   LIN {X -2.697, Y 24.640, Z 108.800}
   LaserStart_Ext()
   LIN {X 5.542, Y 24.640, Z 108.800}
   LaserEnd_Ext()
   LIN {X 5.139, Y 25.640, Z 108.800}
   LaserStart_Ext()
   LIN {X -2.964, Y 25.640, Z 108.800}
   LaserEnd_Ext()
   LIN {X -3.277, Y 26.640, Z 108.800}
   LaserStart_Ext()
   LIN {X 4.736, Y 26.640, Z 108.800}
   LaserEnd_Ext()
   LIN {X 4.333, Y 27.640, Z 108.800}
   LaserStart_Ext()
   LIN {X -3.590, Y 27.640, Z 108.800}
   LaserEnd_Ext()
   LIN {X -3.904, Y 28.640, Z 108.800}
   LaserStart_Ext()
   LIN {X 3.928, Y 28.640, Z 108.800}
   LaserEnd_Ext()
   LIN {X 3.522, Y 29.640, Z 108.800}
   LaserStart_Ext()
   LIN {X -4.217, Y 29.640, Z 108.800}
   LaserEnd_Ext()
   LIN {X -4.535, Y 30.640, Z 108.800}
   LaserStart_Ext()
   LIN {X 3.115, Y 30.640, Z 108.800}
   LaserEnd_Ext()
   LIN {X 2.665, Y 31.640, Z 108.800}
   LaserStart_Ext()
   LIN {X -4.878, Y 31.640, Z 108.800}
   LaserEnd_Ext()
   LIN {X -5.267, Y 32.640, Z 108.800}
   LaserStart_Ext()
   LIN {X 2.196, Y 32.640, Z 108.800}
   LaserEnd_Ext()
   LIN {X 1.727, Y 33.640, Z 108.800}
   LaserStart_Ext()
   LIN {X -5.672, Y 33.640, Z 108.800}
   LaserEnd_Ext()
   LIN {X -6.078, Y 34.640, Z 108.800}
   LaserStart_Ext()
   LIN {X 1.258, Y 34.640, Z 108.800}
   LaserEnd_Ext()
   LIN {X 0.780, Y 35.640, Z 108.800}
   LaserStart_Ext()
   LIN {X -6.479, Y 35.640, Z 108.800}
   LaserEnd_Ext()
   LIN {X -6.928, Y 36.640, Z 108.800}
   LaserStart_Ext()
   LIN {X 0.261, Y 36.640, Z 108.800}
   LaserEnd_Ext()
   LIN {X -0.257, Y 37.640, Z 108.800}
   LaserStart_Ext()
   LIN {X -7.401, Y 37.640, Z 108.800}
   LaserEnd_Ext()
   LIN {X -7.872, Y 38.640, Z 108.800}
   LaserStart_Ext()
   LIN {X -0.776, Y 38.640, Z 108.800}
   LaserEnd_Ext()
   LIN {X -1.330, Y 39.640, Z 108.800}
   LaserStart_Ext()
   LIN {X -8.360, Y 39.640, Z 108.800}
   LaserEnd_Ext()
   LIN {X -8.875, Y 40.640, Z 108.800}
   LaserStart_Ext()
   LIN {X -1.888, Y 40.640, Z 108.800}
   LaserEnd_Ext()
   LIN {X -2.450, Y 41.640, Z 108.800}
   LaserStart_Ext()
   LIN {X -9.405, Y 41.640, Z 108.800}
   LaserEnd_Ext()
   LIN {X -9.750, Y 42.640, Z 108.800}
   LaserStart_Ext()
   LIN {X -3.040, Y 42.640, Z 108.800}
   LaserEnd_Ext()
   LIN {X -3.637, Y 43.640, Z 108.800}
   LaserStart_Ext()
   LIN {X -9.750, Y 43.640, Z 108.800}
   LaserEnd_Ext()
   LIN {X -9.395, Y 44.640, Z 108.800}
   LaserStart_Ext()
   LIN {X -4.259, Y 44.640, Z 108.800}
   LaserEnd_Ext()
   LIN {X -5.251, Y 45.640, Z 108.800}
   LaserStart_Ext()
   LIN {X -8.233, Y 45.640, Z 108.800}
   LaserEnd_Ext()
   LIN {X 1.489, Y -21.393, Z 109.650}
   LaserStart_Ext()
   LIN {X 0.670, Y -20.523, Z 109.650} C_DIS
   LIN {X 0.063, Y -19.874, Z 109.650} C_DIS
   LIN {X -0.221, Y -19.031, Z 109.650} C_DIS
   LIN {X -0.606, Y -17.898, Z 109.650} C_DIS
   LIN {X -0.326, Y -16.414, Z 109.650} C_DIS
   LIN {X -0.042, Y -14.930, Z 109.650} C_DIS
   LIN {X 0.678, Y -14.083, Z 109.650} C_DIS
   LIN {X 1.314, Y -13.320, Z 109.650} C_DIS
   LIN {X 2.671, Y -12.676, Z 109.650} C_DIS
   LIN {X 3.283, Y -12.391, Z 109.650} C_DIS
   LIN {X 3.733, Y -12.383, Z 109.650} C_DIS
   LIN {X 5.327, Y -12.346, Z 109.650} C_DIS
   LIN {X 7.253, Y -13.170, Z 109.650} C_DIS
   LIN {X 8.910, Y -15.135, Z 109.650} C_DIS
   LIN {X 9.327, Y -17.089, Z 109.650} C_DIS
   LIN {X 9.371, Y -17.296, Z 109.650} C_DIS
   LIN {X 9.327, Y -17.466, Z 109.650} C_DIS
   LIN {X 8.781, Y -19.598, Z 109.650} C_DIS
   LIN {X 7.725, Y -20.854, Z 109.650} C_DIS
   LIN {X 7.412, Y -21.228, Z 109.650} C_DIS
   LIN {X 7.138, Y -21.359, Z 109.650} C_DIS
   LIN {X 5.442, Y -22.155, Z 109.650} C_DIS
   LIN {X 3.827, Y -22.190, Z 109.650} C_DIS
   LIN {X 3.393, Y -22.198, Z 109.650} C_DIS
   LIN {X 2.837, Y -21.962, Z 109.650} C_DIS
   LIN {X 1.489, Y -21.393, Z 109.650}
   LaserEnd_Ext()
   LIN {X -4.282, Y -14.760, Z 109.650}
   LaserStart_Ext()
   LIN {X -3.982, Y -13.681, Z 109.650} C_DIS
   LIN {X -3.420, Y -11.591, Z 109.650} C_DIS
   LIN {X -2.903, Y -9.352, Z 109.650} C_DIS
   LIN {X -2.524, Y -7.491, Z 109.650} C_DIS
   LIN {X -1.956, Y -3.894, Z 109.650} C_DIS
   LIN {X -1.776, Y -2.661, Z 109.650} C_DIS
   LIN {X -1.617, Y 0.191, Z 109.650} C_DIS
   LIN {X -1.266, Y 6.431, Z 109.650} C_DIS
   LIN {X -1.777, Y 13.863, Z 109.650} C_DIS
   LIN {X -1.992, Y 16.194, Z 109.650} C_DIS
   LIN {X -3.301, Y 22.823, Z 109.650} C_DIS
   LIN {X -3.707, Y 24.598, Z 109.650} C_DIS
   LIN {X -5.619, Y 30.703, Z 109.650} C_DIS
   LIN {X -5.779, Y 31.168, Z 109.650} C_DIS
   LIN {X -6.169, Y 32.130, Z 109.650} C_DIS
   LIN {X -7.286, Y 34.920, Z 109.650} C_DIS
   LIN {X -7.746, Y 35.978, Z 109.650} C_DIS
   LIN {X -8.768, Y 38.129, Z 109.650} C_DIS
   LIN {X -9.086, Y 38.790, Z 109.650} C_DIS
   LIN {X -9.358, Y 39.314, Z 109.650} C_DIS
   LIN {X -9.821, Y 40.210, Z 109.650} C_DIS
   LIN {X -10.040, Y 40.622, Z 109.650} C_DIS
   LIN {X -10.410, Y 41.313, Z 109.650} C_DIS
   LIN {X -10.836, Y 42.563, Z 109.650} C_DIS
   LIN {X -10.879, Y 42.690, Z 109.650} C_DIS
   LIN {X -10.870, Y 42.819, Z 109.650} C_DIS
   LIN {X -10.782, Y 44.291, Z 109.650} C_DIS
   LIN {X -10.019, Y 45.769, Z 109.650} C_DIS
   LIN {X -7.883, Y 47.113, Z 109.650} C_DIS
   LIN {X -6.707, Y 47.131, Z 109.650} C_DIS
   LIN {X -6.141, Y 47.141, Z 109.650} C_DIS
   LIN {X -5.839, Y 47.006, Z 109.650} C_DIS
   LIN {X -4.557, Y 46.429, Z 109.650} C_DIS
   LIN {X -3.571, Y 45.353, Z 109.650} C_DIS
   LIN {X -2.779, Y 44.088, Z 109.650} C_DIS
   LIN {X -2.138, Y 43.021, Z 109.650} C_DIS
   LIN {X -1.888, Y 42.601, Z 109.650} C_DIS
   LIN {X -1.451, Y 41.852, Z 109.650} C_DIS
   LIN {X -1.083, Y 41.197, Z 109.650} C_DIS
   LIN {X 0.229, Y 38.835, Z 109.650} C_DIS
   LIN {X 1.364, Y 36.647, Z 109.650} C_DIS
   LIN {X 1.693, Y 36.009, Z 109.650} C_DIS
   LIN {X 2.317, Y 34.705, Z 109.650} C_DIS
   LIN {X 4.029, Y 31.053, Z 109.650} C_DIS
   LIN {X 4.856, Y 29.019, Z 109.650} C_DIS
   LIN {X 6.708, Y 24.426, Z 109.650} C_DIS
   LIN {X 7.270, Y 22.711, Z 109.650} C_DIS
   LIN {X 9.117, Y 17.082, Z 109.650} C_DIS
   LIN {X 10.101, Y 13.078, Z 109.650} C_DIS
   LIN {X 11.511, Y 7.032, Z 109.650} C_DIS
   LIN {X 12.575, Y 0.012, Z 109.650} C_DIS
   LIN {X 12.770, Y -1.347, Z 109.650} C_DIS
   LIN {X 13.254, Y -7.226, Z 109.650} C_DIS
   LIN {X 13.286, Y -7.628, Z 109.650} C_DIS
   LIN {X 13.318, Y -8.447, Z 109.650} C_DIS
   LIN {X 13.422, Y -11.308, Z 109.650} C_DIS
   LIN {X 13.441, Y -14.201, Z 109.650} C_DIS
   LIN {X 13.437, Y -14.410, Z 109.650} C_DIS
   LIN {X 13.375, Y -17.530, Z 109.650} C_DIS
   LIN {X 13.069, Y -19.048, Z 109.650} C_DIS
   LIN {X 12.783, Y -20.433, Z 109.650} C_DIS
   LIN {X 11.737, Y -22.221, Z 109.650} C_DIS
   LIN {X 11.254, Y -23.037, Z 109.650} C_DIS
   LIN {X 10.165, Y -23.855, Z 109.650} C_DIS
   LIN {X 8.463, Y -25.189, Z 109.650} C_DIS
   LIN {X 8.006, Y -25.498, Z 109.650} C_DIS
   LIN {X 6.965, Y -25.798, Z 109.650} C_DIS
   LIN {X 5.376, Y -26.226, Z 109.650} C_DIS
   LIN {X 4.199, Y -26.145, Z 109.650} C_DIS
   LIN {X 2.023, Y -25.999, Z 109.650} C_DIS
   LIN {X -0.563, Y -24.720, Z 109.650} C_DIS
   LIN {X -1.210, Y -24.412, Z 109.650} C_DIS
   LIN {X -1.616, Y -23.929, Z 109.650} C_DIS
   LIN {X -3.645, Y -21.485, Z 109.650} C_DIS
   LIN {X -4.310, Y -19.072, Z 109.650} C_DIS
   LIN {X -4.638, Y -17.911, Z 109.650} C_DIS
   LIN {X -4.449, Y -16.198, Z 109.650} C_DIS
   LIN {X -4.282, Y -14.760, Z 109.650}
   LaserEnd_Ext()
   LIN {X 11.602, Y -20.471, Z 109.650}
   LaserStart_Ext()
   LIN {X 11.602, Y -0.245, Z 109.650}
   LaserEnd_Ext()
   LIN {X 10.602, Y 6.357, Z 109.650}
   LaserStart_Ext()
   LIN {X 10.602, Y -22.175, Z 109.650}
   LaserEnd_Ext()
   LIN {X 9.602, Y -23.027, Z 109.650}
   LaserStart_Ext()
   LIN {X 9.602, Y -20.168, Z 109.650}
   LaserEnd_Ext()
   LIN {X 9.602, Y -14.404, Z 109.650}
   LaserStart_Ext()
   LIN {X 9.602, Y 10.816, Z 109.650}
   LaserEnd_Ext()
   LIN {X 8.602, Y 14.989, Z 109.650}
   LaserStart_Ext()
   LIN {X 8.602, Y -13.204, Z 109.650}
   LaserEnd_Ext()
   LIN {X 8.602, Y -21.365, Z 109.650}
   LaserStart_Ext()
   LIN {X 8.602, Y -23.809, Z 109.650}
   LaserEnd_Ext()
   LIN {X 7.602, Y -24.564, Z 109.650}
   LaserStart_Ext()
   LIN {X 7.602, Y -22.245, Z 109.650}
   LaserEnd_Ext()
   LIN {X 7.602, Y -12.232, Z 109.650}
   LaserStart_Ext()
   LIN {X 7.602, Y 18.492, Z 109.650}
   LaserEnd_Ext()
   LIN {X 6.602, Y 21.540, Z 109.650}
   LaserStart_Ext()
   LIN {X 6.602, Y -11.804, Z 109.650}
   LaserEnd_Ext()
   LIN {X 6.602, Y -22.715, Z 109.650}
   LaserStart_Ext()
   LIN {X 6.602, Y -24.861, Z 109.650}
   LaserEnd_Ext()
   LIN {X 5.602, Y -25.130, Z 109.650}
   LaserStart_Ext()
   LIN {X 5.602, Y -23.141, Z 109.650}
   LaserEnd_Ext()
   LIN {X 5.602, Y -11.386, Z 109.650}
   LaserStart_Ext()
   LIN {X 5.602, Y 24.495, Z 109.650}
   LaserEnd_Ext()
   LIN {X 4.602, Y 26.976, Z 109.650}
   LaserStart_Ext()
   LIN {X 4.602, Y -11.363, Z 109.650}
   LaserEnd_Ext()
   LIN {X 4.602, Y -23.174, Z 109.650}
   LaserStart_Ext()
   LIN {X 4.602, Y -25.171, Z 109.650}
   LaserEnd_Ext()
   LIN {X 3.602, Y -25.103, Z 109.650}
   LaserStart_Ext()
   LIN {X 3.602, Y -23.194, Z 109.650}
   LaserEnd_Ext()
   LIN {X 3.602, Y -11.385, Z 109.650}
   LaserStart_Ext()
   LIN {X 3.602, Y 29.449, Z 109.650}
   LaserEnd_Ext()
   LIN {X 2.602, Y 31.741, Z 109.650}
   LaserStart_Ext()
   LIN {X 2.602, Y -11.605, Z 109.650}
   LaserEnd_Ext()
   LIN {X 2.602, Y -22.948, Z 109.650}
   LaserStart_Ext()
   LIN {X 2.602, Y -25.036, Z 109.650}
   LaserEnd_Ext()
   LIN {X 1.602, Y -24.675, Z 109.650}
   LaserStart_Ext()
   LIN {X 1.602, Y -22.526, Z 109.650}
   LaserEnd_Ext()
   LIN {X 1.602, Y -12.077, Z 109.650}
   LaserStart_Ext()
   LIN {X 1.602, Y 33.874, Z 109.650}
   LaserEnd_Ext()
   LIN {X 0.602, Y 35.943, Z 109.650}
   LaserStart_Ext()
   LIN {X 0.602, Y -12.620, Z 109.650}
   LaserEnd_Ext()
   LIN {X 0.602, Y -21.910, Z 109.650}
   LaserStart_Ext()
   LIN {X 0.602, Y -24.181, Z 109.650}
   LaserEnd_Ext()
   LIN {X -0.398, Y -23.691, Z 109.650}
   LaserStart_Ext()
   LIN {X -0.398, Y -20.845, Z 109.650}
   LaserEnd_Ext()
   LIN {X -0.398, Y -13.805, Z 109.650}
   LaserStart_Ext()
   LIN {X -0.398, Y 4.053, Z 109.650}
   LaserEnd_Ext()
   LIN {X -0.398, Y 8.383, Z 109.650}
   LaserStart_Ext()
   LIN {X -0.398, Y 37.873, Z 109.650}
   LaserEnd_Ext()
   LIN {X -1.398, Y 39.705, Z 109.650}
   LaserStart_Ext()
   LIN {X -1.398, Y 18.348, Z 109.650}
   LaserEnd_Ext()
   LIN {X -1.398, Y -6.770, Z 109.650}
   LaserStart_Ext()
   LIN {X -1.398, Y -16.700, Z 109.650}
   LaserEnd_Ext()
   LIN {X -1.398, Y -18.675, Z 109.650}
   LaserStart_Ext()
   LIN {X -1.398, Y -22.626, Z 109.650}
   LaserEnd_Ext()
   LIN {X -2.398, Y -21.422, Z 109.650}
   LaserStart_Ext()
   LIN {X -2.398, Y -11.608, Z 109.650}
   LaserEnd_Ext()
   LIN {X -2.398, Y 23.362, Z 109.650}
   LaserStart_Ext()
   LIN {X -2.398, Y 41.491, Z 109.650}
   LaserEnd_Ext()
   LIN {X -3.398, Y 43.177, Z 109.650}
   LaserStart_Ext()
   LIN {X -3.398, Y 26.958, Z 109.650}
   LaserEnd_Ext()
   LIN {X -3.398, Y -15.818, Z 109.650}
   LaserStart_Ext()
   LIN {X -3.398, Y -18.623, Z 109.650}
   LaserEnd_Ext()
   LIN {X -4.398, Y 30.150, Z 109.650}
   LaserStart_Ext()
   LIN {X -4.398, Y 44.775, Z 109.650}
   LaserEnd_Ext()
   LIN {X -5.398, Y 45.711, Z 109.650}
   LaserStart_Ext()
   LIN {X -5.398, Y 32.895, Z 109.650}
   LaserEnd_Ext()
   LIN {X -6.398, Y 35.386, Z 109.650}
   LaserStart_Ext()
   LIN {X -6.398, Y 46.137, Z 109.650}
   LaserEnd_Ext()
   LIN {X -7.398, Y 46.120, Z 109.650}
   LaserStart_Ext()
   LIN {X -7.398, Y 37.576, Z 109.650}
   LaserEnd_Ext()
   LIN {X -8.398, Y 39.636, Z 109.650}
   LaserStart_Ext()
   LIN {X -8.398, Y 45.608, Z 109.650}
   LaserEnd_Ext()
   LIN {X -9.398, Y 44.792, Z 109.650}
   LaserStart_Ext()
   LIN {X -9.398, Y 41.541, Z 109.650}
   LaserEnd_Ext()
   LIN {X 9.159, Y -15.876, Z 110.500}
   LaserStart_Ext()
   LIN {X 9.452, Y -17.224, Z 110.500} C_DIS
   LIN {X 8.918, Y -19.313, Z 110.500} C_DIS
   LIN {X 8.863, Y -19.534, Z 110.500} C_DIS
   LIN {X 8.686, Y -19.746, Z 110.500} C_DIS
   LIN {X 7.502, Y -21.161, Z 110.500} C_DIS
   LIN {X 6.049, Y -21.850, Z 110.500} C_DIS
   LIN {X 5.533, Y -22.093, Z 110.500} C_DIS
   LIN {X 4.715, Y -22.110, Z 110.500} C_DIS
   LIN {X 3.485, Y -22.140, Z 110.500} C_DIS
   LIN {X 2.667, Y -21.799, Z 110.500} C_DIS
   LIN {X 1.578, Y -21.339, Z 110.500} C_DIS
   LIN {X 0.585, Y -20.284, Z 110.500} C_DIS
   LIN {X 0.149, Y -19.823, Z 110.500} C_DIS
   LIN {X -0.038, Y -19.279, Z 110.500} C_DIS
   LIN {X -0.524, Y -17.849, Z 110.500} C_DIS
   LIN {X -0.045, Y -15.306, Z 110.500} C_DIS
   LIN {X 0.032, Y -14.881, Z 110.500} C_DIS
   LIN {X 0.198, Y -14.676, Z 110.500} C_DIS
   LIN {X 1.349, Y -13.296, Z 110.500} C_DIS
   LIN {X 2.619, Y -12.693, Z 110.500} C_DIS
   LIN {X 3.324, Y -12.341, Z 110.500} C_DIS
   LIN {X 4.429, Y -12.306, Z 110.500} C_DIS
   LIN {X 5.396, Y -12.284, Z 110.500} C_DIS
   LIN {X 6.103, Y -12.586, Z 110.500} C_DIS
   LIN {X 7.353, Y -13.115, Z 110.500} C_DIS
   LIN {X 8.444, Y -14.415, Z 110.500} C_DIS
   LIN {X 8.985, Y -15.064, Z 110.500} C_DIS
   LIN {X 9.159, Y -15.876, Z 110.500}
   LaserEnd_Ext()
   LIN {X -1.499, Y 1.541, Z 110.500}
   LaserStart_Ext()
   LIN {X -1.737, Y -2.717, Z 110.500} C_DIS
   LIN {X -2.006, Y -4.558, Z 110.500} C_DIS
   LIN {X -2.448, Y -7.354, Z 110.500} C_DIS
   LIN {X -2.950, Y -9.818, Z 110.500} C_DIS
   LIN {X -3.303, Y -11.346, Z 110.500} C_DIS
   LIN {X -4.163, Y -14.551, Z 110.500} C_DIS
   LIN {X -4.207, Y -14.720, Z 110.500} C_DIS
   LIN {X -4.555, Y -17.871, Z 110.500} C_DIS
   LIN {X -3.920, Y -20.117, Z 110.500} C_DIS
   LIN {X -3.554, Y -21.444, Z 110.500} C_DIS
   LIN {X -2.439, Y -22.788, Z 110.500} C_DIS
   LIN {X -1.110, Y -24.364, Z 110.500} C_DIS
   LIN {X 1.005, Y -25.374, Z 110.500} C_DIS
   LIN {X 2.207, Y -25.968, Z 110.500} C_DIS
   LIN {X 3.218, Y -26.036, Z 110.500} C_DIS
   LIN {X 5.323, Y -26.181, Z 110.500} C_DIS
   LIN {X 7.970, Y -25.468, Z 110.500} C_DIS
   LIN {X 8.082, Y -25.440, Z 110.500} C_DIS
   LIN {X 8.193, Y -25.360, Z 110.500} C_DIS
   LIN {X 11.282, Y -23.039, Z 110.500} C_DIS
   LIN {X 12.767, Y -20.530, Z 110.500} C_DIS
   LIN {X 12.871, Y -20.353, Z 110.500} C_DIS
   LIN {X 12.899, Y -20.216, Z 110.500} C_DIS
   LIN {X 13.458, Y -17.448, Z 110.500} C_DIS
   LIN {X 13.500, Y -15.336, Z 110.500} C_DIS
   LIN {X 13.517, Y -14.186, Z 110.500} C_DIS
   LIN {X 13.501, Y -12.892, Z 110.500} C_DIS
   LIN {X 13.490, Y -11.226, Z 110.500} C_DIS
   LIN {X 13.433, Y -9.655, Z 110.500} C_DIS
   LIN {X 13.356, Y -7.714, Z 110.500} C_DIS
   LIN {X 13.282, Y -6.761, Z 110.500} C_DIS
   LIN {X 12.861, Y -1.648, Z 110.500} C_DIS
   LIN {X 12.481, Y 0.998, Z 110.500} C_DIS
   LIN {X 11.630, Y 6.615, Z 110.500} C_DIS
   LIN {X 9.957, Y 13.790, Z 110.500} C_DIS
   LIN {X 9.207, Y 16.842, Z 110.500} C_DIS
   LIN {X 7.168, Y 23.056, Z 110.500} C_DIS
   LIN {X 6.759, Y 24.303, Z 110.500} C_DIS
   LIN {X 4.724, Y 29.352, Z 110.500} C_DIS
   LIN {X 4.151, Y 30.761, Z 110.500} C_DIS
   LIN {X 2.965, Y 33.290, Z 110.500} C_DIS
   LIN {X 1.589, Y 36.165, Z 110.500} C_DIS
   LIN {X 0.864, Y 37.571, Z 110.500} C_DIS
   LIN {X 0.372, Y 38.520, Z 110.500} C_DIS
   LIN {X -0.995, Y 40.981, Z 110.500} C_DIS
   LIN {X -1.347, Y 41.611, Z 110.500} C_DIS
   LIN {X -1.430, Y 41.753, Z 110.500} C_DIS
   LIN {X -2.007, Y 42.738, Z 110.500} C_DIS
   LIN {X -2.678, Y 43.851, Z 110.500} C_DIS
   LIN {X -2.846, Y 44.130, Z 110.500} C_DIS
   LIN {X -2.955, Y 44.305, Z 110.500} C_DIS
   LIN {X -3.637, Y 45.385, Z 110.500} C_DIS
   LIN {X -4.589, Y 46.422, Z 110.500} C_DIS
   LIN {X -4.722, Y 46.507, Z 110.500} C_DIS
   LIN {X -6.216, Y 47.174, Z 110.500} C_DIS
   LIN {X -7.216, Y 47.157, Z 110.500} C_DIS
   LIN {X -7.957, Y 47.142, Z 110.500} C_DIS
   LIN {X -8.723, Y 46.647, Z 110.500} C_DIS
   LIN {X -10.111, Y 45.769, Z 110.500} C_DIS
   LIN {X -10.775, Y 44.442, Z 110.500} C_DIS
   LIN {X -10.858, Y 44.280, Z 110.500} C_DIS
   LIN {X -10.869, Y 44.092, Z 110.500} C_DIS
   LIN {X -10.943, Y 42.710, Z 110.500} C_DIS
   LIN {X -10.569, Y 41.627, Z 110.500} C_DIS
   LIN {X -10.470, Y 41.336, Z 110.500} C_DIS
   LIN {X -10.275, Y 40.974, Z 110.500} C_DIS
   LIN {X -9.878, Y 40.235, Z 110.500} C_DIS
   LIN {X -9.556, Y 39.620, Z 110.500} C_DIS
   LIN {X -9.140, Y 38.817, Z 110.500} C_DIS
   LIN {X -8.066, Y 36.588, Z 110.500} C_DIS
   LIN {X -7.929, Y 36.303, Z 110.500} C_DIS
   LIN {X -7.870, Y 36.182, Z 110.500} C_DIS
   LIN {X -7.812, Y 36.049, Z 110.500} C_DIS
   LIN {X -7.115, Y 34.448, Z 110.500} C_DIS
   LIN {X -5.823, Y 31.221, Z 110.500} C_DIS
   LIN {X -5.719, Y 30.956, Z 110.500} C_DIS
   LIN {X -5.174, Y 29.215, Z 110.500} C_DIS
   LIN {X -3.623, Y 24.264, Z 110.500} C_DIS
   LIN {X -3.378, Y 23.191, Z 110.500} C_DIS
   LIN {X -1.948, Y 15.945, Z 110.500} C_DIS
   LIN {X -1.801, Y 14.356, Z 110.500} C_DIS
   LIN {X -1.239, Y 6.181, Z 110.500} C_DIS
   LIN {X -1.499, Y 1.541, Z 110.500}
   LaserEnd_Ext()
   LIN {X -8.631, Y 45.522, Z 110.500}
   LaserStart_Ext()
   LIN {X -5.120, Y 45.522, Z 110.500}
   LaserEnd_Ext()
   LIN {X -4.275, Y 44.522, Z 110.500}
   LaserStart_Ext()
   LIN {X -9.617, Y 44.522, Z 110.500}
   LaserEnd_Ext()
   LIN {X -9.898, Y 43.522, Z 110.500}
   LaserStart_Ext()
   LIN {X -3.647, Y 43.522, Z 110.500}
   LaserEnd_Ext()
   LIN {X -3.044, Y 42.522, Z 110.500}
   LaserStart_Ext()
   LIN {X -9.820, Y 42.522, Z 110.500}
   LaserEnd_Ext()
   LIN {X -9.434, Y 41.522, Z 110.500}
   LaserStart_Ext()
   LIN {X -2.454, Y 41.522, Z 110.500}
   LaserEnd_Ext()
   LIN {X -1.884, Y 40.522, Z 110.500}
   LaserStart_Ext()
   LIN {X -8.899, Y 40.522, Z 110.500}
   LaserEnd_Ext()
   LIN {X -8.379, Y 39.522, Z 110.500}
   LaserStart_Ext()
   LIN {X -1.328, Y 39.522, Z 110.500}
   LaserEnd_Ext()
   LIN {X -0.773, Y 38.522, Z 110.500}
   LaserStart_Ext()
   LIN {X -7.888, Y 38.522, Z 110.500}
   LaserEnd_Ext()
   LIN {X -7.406, Y 37.522, Z 110.500}
   LaserStart_Ext()
   LIN {X -0.236, Y 37.522, Z 110.500}
   LaserEnd_Ext()
   LIN {X 0.280, Y 36.522, Z 110.500}
   LaserStart_Ext()
   LIN {X -6.927, Y 36.522, Z 110.500}
   LaserEnd_Ext()
   LIN {X -6.492, Y 35.522, Z 110.500}
   LaserStart_Ext()
   LIN {X 0.788, Y 35.522, Z 110.500}
   LaserEnd_Ext()
   LIN {X 1.267, Y 34.522, Z 110.500}
   LaserStart_Ext()
   LIN {X -6.067, Y 34.522, Z 110.500}
   LaserEnd_Ext()
   LIN {X -5.667, Y 33.522, Z 110.500}
   LaserStart_Ext()
   LIN {X 1.745, Y 33.522, Z 110.500}
   LaserEnd_Ext()
   LIN {X 2.220, Y 32.522, Z 110.500}
   LaserStart_Ext()
   LIN {X -5.267, Y 32.522, Z 110.500}
   LaserEnd_Ext()
   LIN {X -4.867, Y 31.522, Z 110.500}
   LaserStart_Ext()
   LIN {X 2.689, Y 31.522, Z 110.500}
   LaserEnd_Ext()
   LIN {X 3.158, Y 30.522, Z 110.500}
   LaserStart_Ext()
   LIN {X -4.533, Y 30.522, Z 110.500}
   LaserEnd_Ext()
   LIN {X -4.223, Y 29.522, Z 110.500}
   LaserStart_Ext()
   LIN {X 3.575, Y 29.522, Z 110.500}
   LaserEnd_Ext()
   LIN {X 3.980, Y 28.522, Z 110.500}
   LaserStart_Ext()
   LIN {X -3.909, Y 28.522, Z 110.500}
   LaserEnd_Ext()
   LIN {X -3.596, Y 27.522, Z 110.500}
   LaserStart_Ext()
   LIN {X 4.383, Y 27.522, Z 110.500}
   LaserEnd_Ext()
   LIN {X 4.787, Y 26.522, Z 110.500}
   LaserStart_Ext()
   LIN {X -3.283, Y 26.522, Z 110.500}
   LaserEnd_Ext()
   LIN {X -2.969, Y 25.522, Z 110.500}
   LaserStart_Ext()
   LIN {X 5.190, Y 25.522, Z 110.500}
   LaserEnd_Ext()
   LIN {X 5.593, Y 24.522, Z 110.500}
   LaserStart_Ext()
   LIN {X -2.658, Y 24.522, Z 110.500}
   LaserEnd_Ext()
   LIN {X -2.428, Y 23.522, Z 110.500}
   LaserStart_Ext()
   LIN {X 5.963, Y 23.522, Z 110.500}
   LaserEnd_Ext()
   LIN {X 6.291, Y 22.522, Z 110.500}
   LaserStart_Ext()
   LIN {X -2.226, Y 22.522, Z 110.500}
   LaserEnd_Ext()
   LIN {X -2.029, Y 21.522, Z 110.500}
   LaserStart_Ext()
   LIN {X 6.619, Y 21.522, Z 110.500}
   LaserEnd_Ext()
   LIN {X 6.947, Y 20.522, Z 110.500}
   LaserStart_Ext()
   LIN {X -1.832, Y 20.522, Z 110.500}
   LaserEnd_Ext()
   LIN {X -1.634, Y 19.522, Z 110.500}
   LaserStart_Ext()
   LIN {X 7.275, Y 19.522, Z 110.500}
   LaserEnd_Ext()
   LIN {X 7.603, Y 18.522, Z 110.500}
   LaserStart_Ext()
   LIN {X -1.437, Y 18.522, Z 110.500}
   LaserEnd_Ext()
   LIN {X -1.240, Y 17.522, Z 110.500}
   LaserStart_Ext()
   LIN {X 7.931, Y 17.522, Z 110.500}
   LaserEnd_Ext()
   LIN {X 8.256, Y 16.522, Z 110.500}
   LaserStart_Ext()
   LIN {X -1.042, Y 16.522, Z 110.500}
   LaserEnd_Ext()
   LIN {X -0.904, Y 15.522, Z 110.500}
   LaserStart_Ext()
   LIN {X 8.502, Y 15.522, Z 110.500}
   LaserEnd_Ext()
   LIN {X 8.747, Y 14.522, Z 110.500}
   LaserStart_Ext()
   LIN {X -0.812, Y 14.522, Z 110.500}
   LaserEnd_Ext()
   LIN {X -0.741, Y 13.522, Z 110.500}
   LaserStart_Ext()
   LIN {X 8.993, Y 13.522, Z 110.500}
   LaserEnd_Ext()
   LIN {X 9.226, Y 12.522, Z 110.500}
   LaserStart_Ext()
   LIN {X -0.673, Y 12.522, Z 110.500}
   LaserEnd_Ext()
   LIN {X -0.604, Y 11.522, Z 110.500}
   LaserStart_Ext()
   LIN {X 9.459, Y 11.522, Z 110.500}
   LaserEnd_Ext()
   LIN {X 9.692, Y 10.522, Z 110.500}
   LaserStart_Ext()
   LIN {X -0.535, Y 10.522, Z 110.500}
   LaserEnd_Ext()
   LIN {X -0.466, Y 9.522, Z 110.500}
   LaserStart_Ext()
   LIN {X 9.925, Y 9.522, Z 110.500}
   LaserEnd_Ext()
   LIN {X 10.159, Y 8.522, Z 110.500}
   LaserStart_Ext()
   LIN {X -0.397, Y 8.522, Z 110.500}
   LaserEnd_Ext()
   LIN {X -0.329, Y 7.522, Z 110.500}
   LaserStart_Ext()
   LIN {X 10.392, Y 7.522, Z 110.500}
   LaserEnd_Ext()
   LIN {X 10.625, Y 6.522, Z 110.500}
   LaserStart_Ext()
   LIN {X -0.260, Y 6.522, Z 110.500}
   LaserEnd_Ext()
   LIN {X -0.274, Y 5.522, Z 110.500}
   LaserStart_Ext()
   LIN {X 10.784, Y 5.522, Z 110.500}
   LaserEnd_Ext()
   LIN {X 10.936, Y 4.522, Z 110.500}
   LaserStart_Ext()
   LIN {X -0.330, Y 4.522, Z 110.500}
   LaserEnd_Ext()
   LIN {X -0.386, Y 3.522, Z 110.500}
   LaserStart_Ext()
   LIN {X 11.087, Y 3.522, Z 110.500}
   LaserEnd_Ext()
   LIN {X 11.239, Y 2.522, Z 110.500}
   LaserStart_Ext()
   LIN {X -0.443, Y 2.522, Z 110.500}
   LaserEnd_Ext()
   LIN {X -0.499, Y 1.522, Z 110.500}
   LaserStart_Ext()
   LIN {X 11.391, Y 1.522, Z 110.500}
   LaserEnd_Ext()
   LIN {X 11.540, Y 0.522, Z 110.500}
   LaserStart_Ext()
   LIN {X -0.555, Y 0.522, Z 110.500}
   LaserEnd_Ext()
   LIN {X -0.610, Y -0.478, Z 110.500}
   LaserStart_Ext()
   LIN {X 11.683, Y -0.478, Z 110.500}
   LaserEnd_Ext()
   LIN {X 11.826, Y -1.478, Z 110.500}
   LaserStart_Ext()
   LIN {X -0.666, Y -1.478, Z 110.500}
   LaserEnd_Ext()
   LIN {X -0.722, Y -2.478, Z 110.500}
   LaserStart_Ext()
   LIN {X 11.926, Y -2.478, Z 110.500}
   LaserEnd_Ext()
   LIN {X 12.008, Y -3.478, Z 110.500}
   LaserStart_Ext()
   LIN {X -0.838, Y -3.478, Z 110.500}
   LaserEnd_Ext()
   LIN {X -0.984, Y -4.478, Z 110.500}
   LaserStart_Ext()
   LIN {X 12.090, Y -4.478, Z 110.500}
   LaserEnd_Ext()
   LIN {X 12.173, Y -5.478, Z 110.500}
   LaserStart_Ext()
   LIN {X -1.139, Y -5.478, Z 110.500}
   LaserEnd_Ext()
   LIN {X -1.297, Y -6.478, Z 110.500}
   LaserStart_Ext()
   LIN {X 12.255, Y -6.478, Z 110.500}
   LaserEnd_Ext()
   LIN {X 12.335, Y -7.478, Z 110.500}
   LaserStart_Ext()
   LIN {X -1.455, Y -7.478, Z 110.500}
   LaserEnd_Ext()
   LIN {X -1.656, Y -8.478, Z 110.500}
   LaserStart_Ext()
   LIN {X 12.385, Y -8.478, Z 110.500}
   LaserEnd_Ext()
   LIN {X 12.425, Y -9.478, Z 110.500}
   LaserStart_Ext()
   LIN {X -1.860, Y -9.478, Z 110.500}
   LaserEnd_Ext()
   LIN {X -2.076, Y -10.478, Z 110.500}
   LaserStart_Ext()
   LIN {X 12.462, Y -10.478, Z 110.500}
   LaserEnd_Ext()
   LIN {X 12.491, Y -11.478, Z 110.500}
   LaserStart_Ext()
   LIN {X 6.056, Y -11.478, Z 110.500}
   LaserEnd_Ext()
   LIN {X 2.813, Y -11.478, Z 110.500}
   LaserStart_Ext()
   LIN {X -2.307, Y -11.478, Z 110.500}
   LaserEnd_Ext()
   LIN {X -2.571, Y -12.478, Z 110.500}
   LaserStart_Ext()
   LIN {X 0.776, Y -12.478, Z 110.500}
   LaserEnd_Ext()
   LIN {X 8.124, Y -12.478, Z 110.500}
   LaserStart_Ext()
   LIN {X 12.498, Y -12.478, Z 110.500}
   LaserEnd_Ext()
   LIN {X 12.508, Y -13.478, Z 110.500}
   LaserStart_Ext()
   LIN {X 8.963, Y -13.478, Z 110.500}
   LaserEnd_Ext()
   LIN {X -0.105, Y -13.478, Z 110.500}
   LaserStart_Ext()
   LIN {X -2.840, Y -13.478, Z 110.500}
   LaserEnd_Ext()
   LIN {X -3.108, Y -14.478, Z 110.500}
   LaserStart_Ext()
   LIN {X -0.882, Y -14.478, Z 110.500}
   LaserEnd_Ext()
   LIN {X 9.794, Y -14.478, Z 110.500}
   LaserStart_Ext()
   LIN {X 12.513, Y -14.478, Z 110.500}
   LaserEnd_Ext()
   LIN {X 12.497, Y -15.478, Z 110.500}
   LaserStart_Ext()
   LIN {X 10.096, Y -15.478, Z 110.500}
   LaserEnd_Ext()
   LIN {X -1.095, Y -15.478, Z 110.500}
   LaserStart_Ext()
   LIN {X -3.284, Y -15.478, Z 110.500}
   LaserEnd_Ext()
   LIN {X -3.394, Y -16.478, Z 110.500}
   LaserStart_Ext()
   LIN {X -1.284, Y -16.478, Z 110.500}
   LaserEnd_Ext()
   LIN {X 10.313, Y -16.478, Z 110.500}
   LaserStart_Ext()
   LIN {X 12.477, Y -16.478, Z 110.500}
   LaserEnd_Ext()
   LIN {X 12.432, Y -17.478, Z 110.500}
   LaserStart_Ext()
   LIN {X 10.419, Y -17.478, Z 110.500}
   LaserEnd_Ext()
   LIN {X -1.472, Y -17.478, Z 110.500}
   LaserStart_Ext()
   LIN {X -3.505, Y -17.478, Z 110.500}
   LaserEnd_Ext()
   LIN {X -3.344, Y -18.478, Z 110.500}
   LaserStart_Ext()
   LIN {X -1.366, Y -18.478, Z 110.500}
   LaserEnd_Ext()
   LIN {X 10.164, Y -18.478, Z 110.500}
   LaserStart_Ext()
   LIN {X 12.230, Y -18.478, Z 110.500}
   LaserEnd_Ext()
   LIN {X 12.028, Y -19.478, Z 110.500}
   LaserStart_Ext()
   LIN {X 9.908, Y -19.478, Z 110.500}
   LaserEnd_Ext()
   LIN {X -1.027, Y -19.478, Z 110.500}
   LaserStart_Ext()
   LIN {X -3.061, Y -19.478, Z 110.500}
   LaserEnd_Ext()
   LIN {X -2.783, Y -20.478, Z 110.500}
   LaserStart_Ext()
   LIN {X -0.605, Y -20.478, Z 110.500}
   LaserEnd_Ext()
   LIN {X 9.377, Y -20.478, Z 110.500}
   LaserStart_Ext()
   LIN {X 11.636, Y -20.478, Z 110.500}
   LaserEnd_Ext()
   LIN {X 11.044, Y -21.478, Z 110.500}
   LaserStart_Ext()
   LIN {X 8.540, Y -21.478, Z 110.500}
   LaserEnd_Ext()
   LIN {X 0.336, Y -21.478, Z 110.500}
   LaserStart_Ext()
   LIN {X -2.226, Y -21.478, Z 110.500}
   LaserEnd_Ext()
   LIN {X -1.392, Y -22.478, Z 110.500}
   LaserStart_Ext()
   LIN {X 1.706, Y -22.478, Z 110.500}
   LaserEnd_Ext()
   LIN {X 7.058, Y -22.478, Z 110.500}
   LaserStart_Ext()
   LIN {X 10.364, Y -22.478, Z 110.500}
   LaserEnd_Ext()
   LIN {X 9.033, Y -23.478, Z 110.500}
   LaserStart_Ext()
   LIN {X -0.549, Y -23.478, Z 110.500}
   LaserEnd_Ext()
   LIN {X 1.451, Y -24.478, Z 110.500}
   LaserStart_Ext()
   LIN {X 7.702, Y -24.478, Z 110.500}
   LaserEnd_Ext()
   LIN {X 7.425, Y -13.047, Z 111.350}
   LaserStart_Ext()
   LIN {X 8.498, Y -14.326, Z 111.350} C_DIS
   LIN {X 9.062, Y -14.993, Z 111.350} C_DIS
   LIN {X 9.207, Y -15.653, Z 111.350} C_DIS
   LIN {X 9.534, Y -17.152, Z 111.350} C_DIS
   LIN {X 9.252, Y -18.252, Z 111.350} C_DIS
   LIN {X 8.945, Y -19.471, Z 111.350} C_DIS
   LIN {X 7.970, Y -20.641, Z 111.350} C_DIS
   LIN {X 7.591, Y -21.093, Z 111.350} C_DIS
   LIN {X 6.695, Y -21.518, Z 111.350} C_DIS
   LIN {X 5.625, Y -22.029, Z 111.350} C_DIS
   LIN {X 4.909, Y -22.049, Z 111.350} C_DIS
   LIN {X 3.577, Y -22.081, Z 111.350} C_DIS
   LIN {X 1.865, Y -21.367, Z 111.350} C_DIS
   LIN {X 1.668, Y -21.285, Z 111.350} C_DIS
   LIN {X 1.558, Y -21.170, Z 111.350} C_DIS
   LIN {X 0.236, Y -19.773, Z 111.350} C_DIS
   LIN {X -0.438, Y -17.814, Z 111.350} C_DIS
   LIN {X 0.093, Y -14.860, Z 111.350} C_DIS
   LIN {X 1.231, Y -13.456, Z 111.350} C_DIS
   LIN {X 1.385, Y -13.272, Z 111.350} C_DIS
   LIN {X 1.554, Y -13.191, Z 111.350} C_DIS
   LIN {X 3.349, Y -12.294, Z 111.350} C_DIS
   LIN {X 4.926, Y -12.244, Z 111.350} C_DIS
   LIN {X 5.466, Y -12.221, Z 111.350} C_DIS
   LIN {X 6.072, Y -12.475, Z 111.350} C_DIS
   LIN {X 7.425, Y -13.047, Z 111.350}
   LaserEnd_Ext()
   LIN {X 13.275, Y -18.683, Z 111.350}
   LaserStart_Ext()
   LIN {X 13.541, Y -17.366, Z 111.350} C_DIS
   LIN {X 13.559, Y -16.470, Z 111.350} C_DIS
   LIN {X 13.594, Y -14.103, Z 111.350} C_DIS
   LIN {X 13.560, Y -11.441, Z 111.350} C_DIS
   LIN {X 13.558, Y -11.143, Z 111.350} C_DIS
   LIN {X 13.547, Y -10.863, Z 111.350} C_DIS
   LIN {X 13.427, Y -7.800, Z 111.350} C_DIS
   LIN {X 13.309, Y -6.296, Z 111.350} C_DIS
   LIN {X 12.951, Y -1.949, Z 111.350} C_DIS
   LIN {X 12.388, Y 1.984, Z 111.350} C_DIS
   LIN {X 11.749, Y 6.199, Z 111.350} C_DIS
   LIN {X 9.813, Y 14.502, Z 111.350} C_DIS
   LIN {X 9.297, Y 16.602, Z 111.350} C_DIS
   LIN {X 7.066, Y 23.401, Z 111.350} C_DIS
   LIN {X 6.811, Y 24.180, Z 111.350} C_DIS
   LIN {X 4.591, Y 29.685, Z 111.350} C_DIS
   LIN {X 4.272, Y 30.469, Z 111.350} C_DIS
   LIN {X 3.613, Y 31.875, Z 111.350} C_DIS
   LIN {X 1.485, Y 36.321, Z 111.350} C_DIS
   LIN {X 0.500, Y 38.234, Z 111.350} C_DIS
   LIN {X 0.320, Y 38.552, Z 111.350} C_DIS
   LIN {X -1.433, Y 41.691, Z 111.350} C_DIS
   LIN {X -1.993, Y 42.644, Z 111.350} C_DIS
   LIN {X -2.127, Y 42.874, Z 111.350} C_DIS
   LIN {X -2.348, Y 43.240, Z 111.350} C_DIS
   LIN {X -2.915, Y 44.170, Z 111.350} C_DIS
   LIN {X -3.673, Y 45.367, Z 111.350} C_DIS
   LIN {X -3.745, Y 45.464, Z 111.350} C_DIS
   LIN {X -4.705, Y 46.502, Z 111.350} C_DIS
   LIN {X -5.916, Y 47.041, Z 111.350} C_DIS
   LIN {X -6.291, Y 47.206, Z 111.350} C_DIS
   LIN {X -6.898, Y 47.194, Z 111.350} C_DIS
   LIN {X -8.032, Y 47.171, Z 111.350} C_DIS
   LIN {X -10.117, Y 45.822, Z 111.350} C_DIS
   LIN {X -10.205, Y 45.766, Z 111.350} C_DIS
   LIN {X -10.936, Y 44.268, Z 111.350} C_DIS
   LIN {X -10.999, Y 42.891, Z 111.350} C_DIS
   LIN {X -11.007, Y 42.732, Z 111.350} C_DIS
   LIN {X -10.952, Y 42.572, Z 111.350} C_DIS
   LIN {X -10.532, Y 41.358, Z 111.350} C_DIS
   LIN {X -10.156, Y 40.667, Z 111.350} C_DIS
   LIN {X -9.936, Y 40.259, Z 111.350} C_DIS
   LIN {X -9.520, Y 39.464, Z 111.350} C_DIS
   LIN {X -9.194, Y 38.843, Z 111.350} C_DIS
   LIN {X -8.507, Y 37.412, Z 111.350} C_DIS
   LIN {X -7.966, Y 36.308, Z 111.350} C_DIS
   LIN {X -7.428, Y 35.089, Z 111.350} C_DIS
   LIN {X -6.944, Y 33.977, Z 111.350} C_DIS
   LIN {X -6.047, Y 31.734, Z 111.350} C_DIS
   LIN {X -5.730, Y 30.930, Z 111.350} C_DIS
   LIN {X -5.677, Y 30.805, Z 111.350} C_DIS
   LIN {X -4.077, Y 25.645, Z 111.350} C_DIS
   LIN {X -3.540, Y 23.931, Z 111.350} C_DIS
   LIN {X -3.455, Y 23.559, Z 111.350} C_DIS
   LIN {X -1.903, Y 15.695, Z 111.350} C_DIS
   LIN {X -1.825, Y 14.850, Z 111.350} C_DIS
   LIN {X -1.211, Y 5.930, Z 111.350} C_DIS
   LIN {X -1.382, Y 2.891, Z 111.350} C_DIS
   LIN {X -1.698, Y -2.773, Z 111.350} C_DIS
   LIN {X -2.057, Y -5.223, Z 111.350} C_DIS
   LIN {X -2.372, Y -7.216, Z 111.350} C_DIS
   LIN {X -2.996, Y -10.283, Z 111.350} C_DIS
   LIN {X -3.185, Y -11.101, Z 111.350} C_DIS
   LIN {X -3.646, Y -12.818, Z 111.350} C_DIS
   LIN {X -4.128, Y -14.680, Z 111.350} C_DIS
   LIN {X -4.243, Y -15.770, Z 111.350} C_DIS
   LIN {X -4.471, Y -17.832, Z 111.350} C_DIS
   LIN {X -3.530, Y -21.161, Z 111.350} C_DIS
   LIN {X -3.464, Y -21.402, Z 111.350} C_DIS
   LIN {X -3.261, Y -21.646, Z 111.350} C_DIS
   LIN {X -1.010, Y -24.316, Z 111.350} C_DIS
   LIN {X 2.231, Y -25.863, Z 111.350} C_DIS
   LIN {X 2.424, Y -25.942, Z 111.350} C_DIS
   LIN {X 2.850, Y -25.969, Z 111.350} C_DIS
   LIN {X 5.269, Y -26.135, Z 111.350} C_DIS
   LIN {X 6.312, Y -25.855, Z 111.350} C_DIS
   LIN {X 8.089, Y -25.412, Z 111.350} C_DIS
   LIN {X 9.846, Y -24.142, Z 111.350} C_DIS
   LIN {X 11.310, Y -23.042, Z 111.350} C_DIS
   LIN {X 12.112, Y -21.686, Z 111.350} C_DIS
   LIN {X 12.893, Y -20.435, Z 111.350} C_DIS
   LIN {X 13.275, Y -18.683, Z 111.350}
   LaserEnd_Ext()
   LIN {X -9.280, Y 41.149, Z 111.350}
   LaserStart_Ext()
   LIN {X -9.280, Y 45.173, Z 111.350}
   LaserEnd_Ext()
   LIN {X -8.280, Y 45.820, Z 111.350}
   LaserStart_Ext()
   LIN {X -8.280, Y 39.248, Z 111.350}
   LaserEnd_Ext()
   LIN {X -7.280, Y 37.180, Z 111.350}
   LaserStart_Ext()
   LIN {X -7.280, Y 46.186, Z 111.350}
   LaserEnd_Ext()
   LIN {X -6.280, Y 46.108, Z 111.350}
   LaserStart_Ext()
   LIN {X -6.280, Y 34.956, Z 111.350}
   LaserEnd_Ext()
   LIN {X -5.280, Y 32.509, Z 111.350}
   LaserStart_Ext()
   LIN {X -5.280, Y 45.650, Z 111.350}
   LaserEnd_Ext()
   LIN {X -4.280, Y 44.457, Z 111.350}
   LaserStart_Ext()
   LIN {X -4.280, Y 29.676, Z 111.350}
   LaserEnd_Ext()
   LIN {X -3.280, Y -18.369, Z 111.350}
   LaserStart_Ext()
   LIN {X -3.280, Y -16.160, Z 111.350}
   LaserEnd_Ext()
   LIN {X -3.280, Y 26.450, Z 111.350}
   LaserStart_Ext()
   LIN {X -3.280, Y 42.847, Z 111.350}
   LaserEnd_Ext()
   LIN {X -2.280, Y 41.157, Z 111.350}
   LaserStart_Ext()
   LIN {X -2.280, Y 22.769, Z 111.350}
   LaserEnd_Ext()
   LIN {X -2.280, Y -11.587, Z 111.350}
   LaserStart_Ext()
   LIN {X -2.280, Y -21.259, Z 111.350}
   LaserEnd_Ext()
   LIN {X -1.280, Y -22.445, Z 111.350}
   LaserStart_Ext()
   LIN {X -1.280, Y -18.440, Z 111.350}
   LaserEnd_Ext()
   LIN {X -1.280, Y -16.817, Z 111.350}
   LaserStart_Ext()
   LIN {X -1.280, Y -6.714, Z 111.350}
   LaserEnd_Ext()
   LIN {X -1.280, Y 17.703, Z 111.350}
   LaserStart_Ext()
   LIN {X -1.280, Y 39.366, Z 111.350}
   LaserEnd_Ext()
   LIN {X -0.280, Y 37.563, Z 111.350}
   LaserStart_Ext()
   LIN {X -0.280, Y 6.960, Z 111.350}
   LaserEnd_Ext()
   LIN {X -0.280, Y 4.682, Z 111.350}
   LaserStart_Ext()
   LIN {X -0.280, Y -13.732, Z 111.350}
   LaserEnd_Ext()
   LIN {X -0.280, Y -20.682, Z 111.350}
   LaserStart_Ext()
   LIN {X -0.280, Y -23.557, Z 111.350}
   LaserEnd_Ext()
   LIN {X 0.720, Y -24.034, Z 111.350}
   LaserStart_Ext()
   LIN {X 0.720, Y -21.739, Z 111.350}
   LaserEnd_Ext()
   LIN {X 0.720, Y -12.526, Z 111.350}
   LaserStart_Ext()
   LIN {X 0.720, Y 35.603, Z 111.350}
   LaserEnd_Ext()
   LIN {X 1.720, Y 33.514, Z 111.350}
   LaserStart_Ext()
   LIN {X 1.720, Y -11.990, Z 111.350}
   LaserEnd_Ext()
   LIN {X 1.720, Y -22.390, Z 111.350}
   LaserStart_Ext()
   LIN {X 1.720, Y -24.512, Z 111.350}
   LaserEnd_Ext()
   LIN {X 2.720, Y -24.958, Z 111.350}
   LaserStart_Ext()
   LIN {X 2.720, Y -22.807, Z 111.350}
   LaserEnd_Ext()
   LIN {X 2.720, Y -11.490, Z 111.350}
   LaserStart_Ext()
   LIN {X 2.720, Y 31.423, Z 111.350}
   LaserEnd_Ext()
   LIN {X 3.720, Y 29.170, Z 111.350}
   LaserStart_Ext()
   LIN {X 3.720, Y -11.282, Z 111.350}
   LaserEnd_Ext()
   LIN {X 3.720, Y -23.078, Z 111.350}
   LaserStart_Ext()
   LIN {X 3.720, Y -25.026, Z 111.350}
   LaserEnd_Ext()
   LIN {X 4.720, Y -25.095, Z 111.350}
   LaserStart_Ext()
   LIN {X 4.720, Y -23.054, Z 111.350}
   LaserEnd_Ext()
   LIN {X 4.720, Y -11.250, Z 111.350}
   LaserStart_Ext()
   LIN {X 4.720, Y 26.690, Z 111.350}
   LaserEnd_Ext()
   LIN {X 5.720, Y 24.210, Z 111.350}
   LaserStart_Ext()
   LIN {X 5.720, Y -11.255, Z 111.350}
   LaserEnd_Ext()
   LIN {X 5.720, Y -23.024, Z 111.350}
   LaserStart_Ext()
   LIN {X 5.720, Y -24.978, Z 111.350}
   LaserEnd_Ext()
   LIN {X 6.720, Y -24.722, Z 111.350}
   LaserStart_Ext()
   LIN {X 6.720, Y -22.615, Z 111.350}
   LaserEnd_Ext()
   LIN {X 6.720, Y -11.664, Z 111.350}
   LaserStart_Ext()
   LIN {X 6.720, Y 21.247, Z 111.350}
   LaserEnd_Ext()
   LIN {X 7.720, Y 18.199, Z 111.350}
   LaserStart_Ext()
   LIN {X 7.720, Y -12.086, Z 111.350}
   LaserEnd_Ext()
   LIN {X 7.720, Y -22.139, Z 111.350}
   LaserStart_Ext()
   LIN {X 7.720, Y -24.445, Z 111.350}
   LaserEnd_Ext()
   LIN {X 8.720, Y -23.722, Z 111.350}
   LaserStart_Ext()
   LIN {X 8.720, Y -21.303, Z 111.350}
   LaserEnd_Ext()
   LIN {X 8.720, Y -13.035, Z 111.350}
   LaserStart_Ext()
   LIN {X 8.720, Y 14.758, Z 111.350}
   LaserEnd_Ext()
   LIN {X 9.720, Y 10.495, Z 111.350}
   LaserStart_Ext()
   LIN {X 9.720, Y -14.223, Z 111.350}
   LaserEnd_Ext()
   LIN {X 9.720, Y -20.103, Z 111.350}
   LaserStart_Ext()
   LIN {X 9.720, Y -22.986, Z 111.350}
   LaserEnd_Ext()
   LIN {X 10.720, Y -22.075, Z 111.350}
   LaserStart_Ext()
   LIN {X 10.720, Y 6.207, Z 111.350}
   LaserEnd_Ext()
   LIN {X 11.720, Y -0.406, Z 111.350}
   LaserStart_Ext()
   LIN {X 11.720, Y -20.426, Z 111.350}
   LaserEnd_Ext()
   LIN {X -0.089, Y -16.177, Z 112.200}
   LaserStart_Ext()
   LIN {X 0.154, Y -14.839, Z 112.200} C_DIS
   LIN {X 0.790, Y -14.054, Z 112.200} C_DIS
   LIN {X 1.443, Y -13.231, Z 112.200} C_DIS
   LIN {X 2.895, Y -12.486, Z 112.200} C_DIS
   LIN {X 3.374, Y -12.247, Z 112.200} C_DIS
   LIN {X 3.711, Y -12.237, Z 112.200} C_DIS
   LIN {X 5.537, Y -12.158, Z 112.200} C_DIS
   LIN {X 7.422, Y -12.949, Z 112.200} C_DIS
   LIN {X 7.563, Y -13.057, Z 112.200} C_DIS
   LIN {X 9.139, Y -14.921, Z 112.200} C_DIS
   LIN {X 9.582, Y -16.927, Z 112.200} C_DIS
   LIN {X 9.615, Y -17.079, Z 112.200} C_DIS
   LIN {X 9.586, Y -17.191, Z 112.200} C_DIS
   LIN {X 9.028, Y -19.408, Z 112.200} C_DIS
   LIN {X 8.366, Y -20.202, Z 112.200} C_DIS
   LIN {X 7.683, Y -21.025, Z 112.200} C_DIS
   LIN {X 7.081, Y -21.315, Z 112.200} C_DIS
   LIN {X 5.719, Y -21.966, Z 112.200} C_DIS
   LIN {X 3.728, Y -22.021, Z 112.200} C_DIS
   LIN {X 3.594, Y -21.991, Z 112.200} C_DIS
   LIN {X 1.760, Y -21.231, Z 112.200} C_DIS
   LIN {X 0.734, Y -20.156, Z 112.200} C_DIS
   LIN {X 0.324, Y -19.722, Z 112.200} C_DIS
   LIN {X 0.111, Y -19.104, Z 112.200} C_DIS
   LIN {X -0.359, Y -17.751, Z 112.200} C_DIS
   LIN {X -0.089, Y -16.177, Z 112.200}
   LaserEnd_Ext()
   LIN {X -2.034, Y 42.648, Z 112.200}
   LaserStart_Ext()
   LIN {X -2.211, Y 42.944, Z 112.200} C_DIS
   LIN {X -2.842, Y 43.976, Z 112.200} C_DIS
   LIN {X -2.985, Y 44.210, Z 112.200} C_DIS
   LIN {X -3.097, Y 44.387, Z 112.200} C_DIS
   LIN {X -3.782, Y 45.462, Z 112.200} C_DIS
   LIN {X -4.688, Y 46.439, Z 112.200} C_DIS
   LIN {X -4.780, Y 46.537, Z 112.200} C_DIS
   LIN {X -4.962, Y 46.617, Z 112.200} C_DIS
   LIN {X -6.369, Y 47.238, Z 112.200} C_DIS
   LIN {X -7.442, Y 47.215, Z 112.200} C_DIS
   LIN {X -8.109, Y 47.199, Z 112.200} C_DIS
   LIN {X -8.848, Y 46.707, Z 112.200} C_DIS
   LIN {X -10.301, Y 45.760, Z 112.200} C_DIS
   LIN {X -10.887, Y 44.517, Z 112.200} C_DIS
   LIN {X -11.015, Y 44.255, Z 112.200} C_DIS
   LIN {X -11.028, Y 43.957, Z 112.200} C_DIS
   LIN {X -11.055, Y 42.641, Z 112.200} C_DIS
   LIN {X -10.677, Y 41.620, Z 112.200} C_DIS
   LIN {X -10.594, Y 41.380, Z 112.200} C_DIS
   LIN {X -10.441, Y 41.099, Z 112.200} C_DIS
   LIN {X -9.996, Y 40.282, Z 112.200} C_DIS
   LIN {X -9.522, Y 39.384, Z 112.200} C_DIS
   LIN {X -9.251, Y 38.868, Z 112.200} C_DIS
   LIN {X -9.084, Y 38.522, Z 112.200} C_DIS
   LIN {X -8.063, Y 36.435, Z 112.200} C_DIS
   LIN {X -7.045, Y 34.129, Z 112.200} C_DIS
   LIN {X -6.774, Y 33.505, Z 112.200} C_DIS
   LIN {X -6.270, Y 32.247, Z 112.200} C_DIS
   LIN {X -5.742, Y 30.903, Z 112.200} C_DIS
   LIN {X -5.652, Y 30.695, Z 112.200} C_DIS
   LIN {X -3.580, Y 24.012, Z 112.200} C_DIS
   LIN {X -3.472, Y 23.657, Z 112.200} C_DIS
   LIN {X -2.223, Y 17.292, Z 112.200} C_DIS
   LIN {X -1.858, Y 15.446, Z 112.200} C_DIS
   LIN {X -1.849, Y 15.344, Z 112.200} C_DIS
   LIN {X -1.184, Y 5.679, Z 112.200} C_DIS
   LIN {X -1.265, Y 4.241, Z 112.200} C_DIS
   LIN {X -1.660, Y -2.829, Z 112.200} C_DIS
   LIN {X -2.107, Y -5.887, Z 112.200} C_DIS
   LIN {X -2.295, Y -7.078, Z 112.200} C_DIS
   LIN {X -3.042, Y -10.748, Z 112.200} C_DIS
   LIN {X -3.067, Y -10.857, Z 112.200} C_DIS
   LIN {X -3.128, Y -11.084, Z 112.200} C_DIS
   LIN {X -4.050, Y -14.640, Z 112.200} C_DIS
   LIN {X -4.269, Y -16.721, Z 112.200} C_DIS
   LIN {X -4.387, Y -17.793, Z 112.200} C_DIS
   LIN {X -3.801, Y -19.868, Z 112.200} C_DIS
   LIN {X -3.369, Y -21.360, Z 112.200} C_DIS
   LIN {X -2.639, Y -22.219, Z 112.200} C_DIS
   LIN {X -0.911, Y -24.269, Z 112.200} C_DIS
   LIN {X 1.193, Y -25.273, Z 112.200} C_DIS
   LIN {X 2.853, Y -25.947, Z 112.200} C_DIS
   LIN {X 4.776, Y -26.069, Z 112.200} C_DIS
   LIN {X 5.224, Y -26.087, Z 112.200} C_DIS
   LIN {X 5.526, Y -26.015, Z 112.200} C_DIS
   LIN {X 5.839, Y -25.946, Z 112.200} C_DIS
   LIN {X 8.096, Y -25.384, Z 112.200} C_DIS
   LIN {X 11.107, Y -23.207, Z 112.200} C_DIS
   LIN {X 11.329, Y -23.053, Z 112.200} C_DIS
   LIN {X 11.398, Y -22.957, Z 112.200} C_DIS
   LIN {X 12.907, Y -20.538, Z 112.200} C_DIS
   LIN {X 13.539, Y -17.642, Z 112.200} C_DIS
   LIN {X 13.625, Y -17.284, Z 112.200} C_DIS
   LIN {X 13.629, Y -16.818, Z 112.200} C_DIS
   LIN {X 13.670, Y -14.020, Z 112.200} C_DIS
   LIN {X 13.645, Y -12.045, Z 112.200} C_DIS
   LIN {X 13.628, Y -11.059, Z 112.200} C_DIS
   LIN {X 13.580, Y -9.981, Z 112.200} C_DIS
   LIN {X 13.497, Y -7.886, Z 112.200} C_DIS
   LIN {X 13.337, Y -5.831, Z 112.200} C_DIS
   LIN {X 13.042, Y -2.250, Z 112.200} C_DIS
   LIN {X 12.294, Y 2.970, Z 112.200} C_DIS
   LIN {X 11.868, Y 5.783, Z 112.200} C_DIS
   LIN {X 9.669, Y 15.214, Z 112.200} C_DIS
   LIN {X 9.386, Y 16.363, Z 112.200} C_DIS
   LIN {X 6.963, Y 23.746, Z 112.200} C_DIS
   LIN {X 6.862, Y 24.056, Z 112.200} C_DIS
   LIN {X 4.458, Y 30.019, Z 112.200} C_DIS
   LIN {X 4.394, Y 30.177, Z 112.200} C_DIS
   LIN {X 4.261, Y 30.461, Z 112.200} C_DIS
   LIN {X 1.382, Y 36.477, Z 112.200} C_DIS
   LIN {X 0.576, Y 38.041, Z 112.200} C_DIS
   LIN {X -0.372, Y 39.718, Z 112.200} C_DIS
   LIN {X -1.518, Y 41.771, Z 112.200} C_DIS
   LIN {X -2.034, Y 42.648, Z 112.200}
   LaserEnd_Ext()
   LIN {X 7.806, Y -24.360, Z 112.200}
   LaserStart_Ext()
   LIN {X 1.603, Y -24.360, Z 112.200}
   LaserEnd_Ext()
   LIN {X -0.369, Y -23.360, Z 112.200}
   LaserStart_Ext()
   LIN {X 9.189, Y -23.360, Z 112.200}
   LaserEnd_Ext()
   LIN {X 10.574, Y -22.360, Z 112.200}
   LaserStart_Ext()
   LIN {X 7.214, Y -22.360, Z 112.200}
   LaserEnd_Ext()
   LIN {X 1.873, Y -22.360, Z 112.200}
   LaserStart_Ext()
   LIN {X -1.212, Y -22.360, Z 112.200}
   LaserEnd_Ext()
   LIN {X -2.056, Y -21.360, Z 112.200}
   LaserStart_Ext()
   LIN {X 0.501, Y -21.360, Z 112.200}
   LaserEnd_Ext()
   LIN {X 8.704, Y -21.360, Z 112.200}
   LaserStart_Ext()
   LIN {X 11.215, Y -21.360, Z 112.200}
   LaserEnd_Ext()
   LIN {X 11.839, Y -20.360, Z 112.200}
   LaserStart_Ext()
   LIN {X 9.536, Y -20.360, Z 112.200}
   LaserEnd_Ext()
   LIN {X -0.445, Y -20.360, Z 112.200}
   LaserStart_Ext()
   LIN {X -2.617, Y -20.360, Z 112.200}
   LaserEnd_Ext()
   LIN {X -2.905, Y -19.360, Z 112.200}
   LaserStart_Ext()
   LIN {X -0.859, Y -19.360, Z 112.200}
   LaserEnd_Ext()
   LIN {X 10.071, Y -19.360, Z 112.200}
   LaserStart_Ext()
   LIN {X 12.140, Y -19.360, Z 112.200}
   LaserEnd_Ext()
   LIN {X 12.359, Y -18.360, Z 112.200}
   LaserStart_Ext()
   LIN {X 10.323, Y -18.360, Z 112.200}
   LaserEnd_Ext()
   LIN {X -1.206, Y -18.360, Z 112.200}
   LaserStart_Ext()
   LIN {X -3.187, Y -18.360, Z 112.200}
   LaserEnd_Ext()
   LIN {X -3.333, Y -17.360, Z 112.200}
   LaserStart_Ext()
   LIN {X -1.306, Y -17.360, Z 112.200}
   LaserEnd_Ext()
   LIN {X 10.575, Y -17.360, Z 112.200}
   LaserStart_Ext()
   LIN {X 12.578, Y -17.360, Z 112.200}
   LaserEnd_Ext()
   LIN {X 12.636, Y -16.360, Z 112.200}
   LaserStart_Ext()
   LIN {X 10.481, Y -16.360, Z 112.200}
   LaserEnd_Ext()
   LIN {X -1.135, Y -16.360, Z 112.200}
   LaserStart_Ext()
   LIN {X -3.225, Y -16.360, Z 112.200}
   LaserEnd_Ext()
   LIN {X -3.120, Y -15.360, Z 112.200}
   LaserStart_Ext()
   LIN {X -0.957, Y -15.360, Z 112.200}
   LaserEnd_Ext()
   LIN {X 10.260, Y -15.360, Z 112.200}
   LaserStart_Ext()
   LIN {X 12.650, Y -15.360, Z 112.200}
   LaserEnd_Ext()
   LIN {X 12.665, Y -14.360, Z 112.200}
   LaserStart_Ext()
   LIN {X 9.966, Y -14.360, Z 112.200}
   LaserEnd_Ext()
   LIN {X -0.722, Y -14.360, Z 112.200}
   LaserStart_Ext()
   LIN {X -2.944, Y -14.360, Z 112.200}
   LaserEnd_Ext()
   LIN {X -2.685, Y -13.360, Z 112.200}
   LaserStart_Ext()
   LIN {X 0.064, Y -13.360, Z 112.200}
   LaserEnd_Ext()
   LIN {X 9.129, Y -13.360, Z 112.200}
   LaserStart_Ext()
   LIN {X 12.662, Y -13.360, Z 112.200}
   LaserEnd_Ext()
   LIN {X 12.649, Y -12.360, Z 112.200}
   LaserStart_Ext()
   LIN {X 8.282, Y -12.360, Z 112.200}
   LaserEnd_Ext()
   LIN {X 0.953, Y -12.360, Z 112.200}
   LaserStart_Ext()
   LIN {X -2.426, Y -12.360, Z 112.200}
   LaserEnd_Ext()
   LIN {X -2.167, Y -11.360, Z 112.200}
   LaserStart_Ext()
   LIN {X 2.912, Y -11.360, Z 112.200}
   LaserEnd_Ext()
   LIN {X 6.221, Y -11.360, Z 112.200}
   LaserStart_Ext()
   LIN {X 12.633, Y -11.360, Z 112.200}
   LaserEnd_Ext()
   LIN {X 12.596, Y -10.360, Z 112.200}
   LaserStart_Ext()
   LIN {X -1.943, Y -10.360, Z 112.200}
   LaserEnd_Ext()
   LIN {X -1.739, Y -9.360, Z 112.200}
   LaserStart_Ext()
   LIN {X 12.555, Y -9.360, Z 112.200}
   LaserEnd_Ext()
   LIN {X 12.515, Y -8.360, Z 112.200}
   LaserStart_Ext()
   LIN {X -1.536, Y -8.360, Z 112.200}
   LaserEnd_Ext()
   LIN {X -1.332, Y -7.360, Z 112.200}
   LaserStart_Ext()
   LIN {X 12.453, Y -7.360, Z 112.200}
   LaserEnd_Ext()
   LIN {X 12.375, Y -6.360, Z 112.200}
   LaserStart_Ext()
   LIN {X -1.169, Y -6.360, Z 112.200}
   LaserEnd_Ext()
   LIN {X -1.019, Y -5.360, Z 112.200}
   LaserStart_Ext()
   LIN {X 12.295, Y -5.360, Z 112.200}
   LaserEnd_Ext()
   LIN {X 12.213, Y -4.360, Z 112.200}
   LaserStart_Ext()
   LIN {X -0.873, Y -4.360, Z 112.200}
   LaserEnd_Ext()
   LIN {X -0.727, Y -3.360, Z 112.200}
   LaserStart_Ext()
   LIN {X 12.130, Y -3.360, Z 112.200}
   LaserEnd_Ext()
   LIN {X 12.048, Y -2.360, Z 112.200}
   LaserStart_Ext()
   LIN {X -0.632, Y -2.360, Z 112.200}
   LaserEnd_Ext()
   LIN {X -0.576, Y -1.360, Z 112.200}
   LaserStart_Ext()
   LIN {X 11.904, Y -1.360, Z 112.200}
   LaserEnd_Ext()
   LIN {X 11.761, Y -0.360, Z 112.200}
   LaserStart_Ext()
   LIN {X -0.520, Y -0.360, Z 112.200}
   LaserEnd_Ext()
   LIN {X -0.464, Y 0.640, Z 112.200}
   LaserStart_Ext()
   LIN {X 11.618, Y 0.640, Z 112.200}
   LaserEnd_Ext()
   LIN {X 11.474, Y 1.640, Z 112.200}
   LaserStart_Ext()
   LIN {X -0.408, Y 1.640, Z 112.200}
   LaserEnd_Ext()
   LIN {X -0.353, Y 2.640, Z 112.200}
   LaserStart_Ext()
   LIN {X 11.331, Y 2.640, Z 112.200}
   LaserEnd_Ext()
   LIN {X 11.181, Y 3.640, Z 112.200}
   LaserStart_Ext()
   LIN {X -0.297, Y 3.640, Z 112.200}
   LaserEnd_Ext()
   LIN {X -0.241, Y 4.640, Z 112.200}
   LaserStart_Ext()
   LIN {X 11.029, Y 4.640, Z 112.200}
   LaserEnd_Ext()
   LIN {X 10.874, Y 5.640, Z 112.200}
   LaserStart_Ext()
   LIN {X -0.186, Y 5.640, Z 112.200}
   LaserEnd_Ext()
   LIN {X -0.248, Y 6.640, Z 112.200}
   LaserStart_Ext()
   LIN {X 10.641, Y 6.640, Z 112.200}
   LaserEnd_Ext()
   LIN {X 10.408, Y 7.640, Z 112.200}
   LaserStart_Ext()
   LIN {X -0.317, Y 7.640, Z 112.200}
   LaserEnd_Ext()
   LIN {X -0.385, Y 8.640, Z 112.200}
   LaserStart_Ext()
   LIN {X 10.175, Y 8.640, Z 112.200}
   LaserEnd_Ext()
   LIN {X 9.941, Y 9.640, Z 112.200}
   LaserStart_Ext()
   LIN {X -0.454, Y 9.640, Z 112.200}
   LaserEnd_Ext()
   LIN {X -0.523, Y 10.640, Z 112.200}
   LaserStart_Ext()
   LIN {X 9.708, Y 10.640, Z 112.200}
   LaserEnd_Ext()
   LIN {X 9.475, Y 11.640, Z 112.200}
   LaserStart_Ext()
   LIN {X -0.592, Y 11.640, Z 112.200}
   LaserEnd_Ext()
   LIN {X -0.661, Y 12.640, Z 112.200}
   LaserStart_Ext()
   LIN {X 9.242, Y 12.640, Z 112.200}
   LaserEnd_Ext()
   LIN {X 9.009, Y 13.640, Z 112.200}
   LaserStart_Ext()
   LIN {X -0.729, Y 13.640, Z 112.200}
   LaserEnd_Ext()
   LIN {X -0.798, Y 14.640, Z 112.200}
   LaserStart_Ext()
   LIN {X 8.776, Y 14.640, Z 112.200}
   LaserEnd_Ext()
   LIN {X 8.534, Y 15.640, Z 112.200}
   LaserStart_Ext()
   LIN {X -0.877, Y 15.640, Z 112.200}
   LaserEnd_Ext()
   LIN {X -1.075, Y 16.640, Z 112.200}
   LaserStart_Ext()
   LIN {X 8.243, Y 16.640, Z 112.200}
   LaserEnd_Ext()
   LIN {X 7.915, Y 17.640, Z 112.200}
   LaserStart_Ext()
   LIN {X -1.272, Y 17.640, Z 112.200}
   LaserEnd_Ext()
   LIN {X -1.468, Y 18.640, Z 112.200}
   LaserStart_Ext()
   LIN {X 7.586, Y 18.640, Z 112.200}
   LaserEnd_Ext()
   LIN {X 7.258, Y 19.640, Z 112.200}
   LaserStart_Ext()
   LIN {X -1.664, Y 19.640, Z 112.200}
   LaserEnd_Ext()
   LIN {X -1.860, Y 20.640, Z 112.200}
   LaserStart_Ext()
   LIN {X 6.930, Y 20.640, Z 112.200}
   LaserEnd_Ext()
   LIN {X 6.602, Y 21.640, Z 112.200}
   LaserStart_Ext()
   LIN {X -2.057, Y 21.640, Z 112.200}
   LaserEnd_Ext()
   LIN {X -2.253, Y 22.640, Z 112.200}
   LaserStart_Ext()
   LIN {X 6.274, Y 22.640, Z 112.200}
   LaserEnd_Ext()
   LIN {X 5.946, Y 23.640, Z 112.200}
   LaserStart_Ext()
   LIN {X -2.449, Y 23.640, Z 112.200}
   LaserEnd_Ext()
   LIN {X -2.728, Y 24.640, Z 112.200}
   LaserStart_Ext()
   LIN {X 5.548, Y 24.640, Z 112.200}
   LaserEnd_Ext()
   LIN {X 5.145, Y 25.640, Z 112.200}
   LaserStart_Ext()
   LIN {X -3.038, Y 25.640, Z 112.200}
   LaserEnd_Ext()
   LIN {X -3.348, Y 26.640, Z 112.200}
   LaserStart_Ext()
   LIN {X 4.742, Y 26.640, Z 112.200}
   LaserEnd_Ext()
   LIN {X 4.339, Y 27.640, Z 112.200}
   LaserStart_Ext()
   LIN {X -3.658, Y 27.640, Z 112.200}
   LaserEnd_Ext()
   LIN {X -3.968, Y 28.640, Z 112.200}
   LaserStart_Ext()
   LIN {X 3.936, Y 28.640, Z 112.200}
   LaserEnd_Ext()
   LIN {X 3.532, Y 29.640, Z 112.200}
   LaserStart_Ext()
   LIN {X -4.278, Y 29.640, Z 112.200}
   LaserEnd_Ext()
   LIN {X -4.588, Y 30.640, Z 112.200}
   LaserStart_Ext()
   LIN {X 3.066, Y 30.640, Z 112.200}
   LaserEnd_Ext()
   LIN {X 2.588, Y 31.640, Z 112.200}
   LaserStart_Ext()
   LIN {X -4.957, Y 31.640, Z 112.200}
   LaserEnd_Ext()
   LIN {X -5.350, Y 32.640, Z 112.200}
   LaserStart_Ext()
   LIN {X 2.109, Y 32.640, Z 112.200}
   LaserEnd_Ext()
   LIN {X 1.631, Y 33.640, Z 112.200}
   LaserStart_Ext()
   LIN {X -5.750, Y 33.640, Z 112.200}
   LaserEnd_Ext()
   LIN {X -6.177, Y 34.640, Z 112.200}
   LaserStart_Ext()
   LIN {X 1.152, Y 34.640, Z 112.200}
   LaserEnd_Ext()
   LIN {X 0.674, Y 35.640, Z 112.200}
   LaserStart_Ext()
   LIN {X -6.619, Y 35.640, Z 112.200}
   LaserEnd_Ext()
   LIN {X -7.060, Y 36.640, Z 112.200}
   LaserStart_Ext()
   LIN {X 0.173, Y 36.640, Z 112.200}
   LaserEnd_Ext()
   LIN {X -0.346, Y 37.640, Z 112.200}
   LaserStart_Ext()
   LIN {X -7.539, Y 37.640, Z 112.200}
   LaserEnd_Ext()
   LIN {X -8.029, Y 38.640, Z 112.200}
   LaserStart_Ext()
   LIN {X -0.911, Y 38.640, Z 112.200}
   LaserEnd_Ext()
   LIN {X -1.474, Y 39.640, Z 112.200}
   LaserStart_Ext()
   LIN {X -8.526, Y 39.640, Z 112.200}
   LaserEnd_Ext()
   LIN {X -9.055, Y 40.640, Z 112.200}
   LaserStart_Ext()
   LIN {X -2.032, Y 40.640, Z 112.200}
   LaserEnd_Ext()
   LIN {X -2.601, Y 41.640, Z 112.200}
   LaserStart_Ext()
   LIN {X -9.597, Y 41.640, Z 112.200}
   LaserEnd_Ext()
   LIN {X -9.988, Y 42.640, Z 112.200}
   LaserStart_Ext()
   LIN {X -3.198, Y 42.640, Z 112.200}
   LaserEnd_Ext()
   LIN {X -3.809, Y 43.640, Z 112.200}
   LaserStart_Ext()
   LIN {X -10.035, Y 43.640, Z 112.200}
   LaserEnd_Ext()
   LIN {X -9.723, Y 44.640, Z 112.200}
   LaserStart_Ext()
   LIN {X -4.443, Y 44.640, Z 112.200}
   LaserEnd_Ext()
   LIN {X -5.311, Y 45.640, Z 112.200}
   LaserStart_Ext()
   LIN {X -8.654, Y 45.640, Z 112.200}
   LaserEnd_Ext()
   LIN {X 9.217, Y -14.849, Z 113.050}
   LaserStart_Ext()
   LIN {X 9.381, Y -15.596, Z 113.050} C_DIS
   LIN {X 9.699, Y -17.006, Z 113.050} C_DIS
   LIN {X 9.489, Y -17.846, Z 113.050} C_DIS
   LIN {X 9.110, Y -19.348, Z 113.050} C_DIS
   LIN {X 8.734, Y -19.802, Z 113.050} C_DIS
   LIN {X 7.775, Y -20.957, Z 113.050} C_DIS
   LIN {X 6.039, Y -21.794, Z 113.050} C_DIS
   LIN {X 5.812, Y -21.902, Z 113.050} C_DIS
   LIN {X 5.458, Y -21.912, Z 113.050} C_DIS
   LIN {X 3.765, Y -21.964, Z 113.050} C_DIS
   LIN {X 2.670, Y -21.516, Z 113.050} C_DIS
   LIN {X 1.852, Y -21.177, Z 113.050} C_DIS
   LIN {X 1.039, Y -20.324, Z 113.050} C_DIS
   LIN {X 0.412, Y -19.671, Z 113.050} C_DIS
   LIN {X 0.113, Y -18.818, Z 113.050} C_DIS
   LIN {X -0.275, Y -17.701, Z 113.050} C_DIS
   LIN {X 0.123, Y -15.377, Z 113.050} C_DIS
   LIN {X 0.204, Y -14.855, Z 113.050} C_DIS
   LIN {X 0.400, Y -14.582, Z 113.050} C_DIS
   LIN {X 1.505, Y -13.187, Z 113.050} C_DIS
   LIN {X 2.635, Y -12.608, Z 113.050} C_DIS
   LIN {X 3.434, Y -12.192, Z 113.050} C_DIS
   LIN {X 4.678, Y -12.135, Z 113.050} C_DIS
   LIN {X 5.608, Y -12.095, Z 113.050} C_DIS
   LIN {X 6.271, Y -12.373, Z 113.050} C_DIS
   LIN {X 7.571, Y -12.911, Z 113.050} C_DIS
   LIN {X 8.713, Y -14.254, Z 113.050} C_DIS
   LIN {X 9.217, Y -14.849, Z 113.050}
   LaserEnd_Ext()
   LIN {X -8.905, Y 38.085, Z 113.050}
   LaserStart_Ext()
   LIN {X -9.308, Y 38.892, Z 113.050} C_DIS
   LIN {X -9.952, Y 40.104, Z 113.050} C_DIS
   LIN {X -10.058, Y 40.304, Z 113.050} C_DIS
   LIN {X -10.130, Y 40.438, Z 113.050} C_DIS
   LIN {X -10.658, Y 41.400, Z 113.050} C_DIS
   LIN {X -11.066, Y 42.456, Z 113.050} C_DIS
   LIN {X -11.103, Y 42.707, Z 113.050} C_DIS
   LIN {X -11.100, Y 44.216, Z 113.050} C_DIS
   LIN {X -10.441, Y 45.657, Z 113.050} C_DIS
   LIN {X -10.398, Y 45.753, Z 113.050} C_DIS
   LIN {X -10.223, Y 45.871, Z 113.050} C_DIS
   LIN {X -8.188, Y 47.226, Z 113.050} C_DIS
   LIN {X -6.972, Y 47.256, Z 113.050} C_DIS
   LIN {X -6.447, Y 47.269, Z 113.050} C_DIS
   LIN {X -6.141, Y 47.136, Z 113.050} C_DIS
   LIN {X -4.858, Y 46.571, Z 113.050} C_DIS
   LIN {X -3.870, Y 45.518, Z 113.050} C_DIS
   LIN {X -3.056, Y 44.249, Z 113.050} C_DIS
   LIN {X -2.483, Y 43.318, Z 113.050} C_DIS
   LIN {X -2.279, Y 42.984, Z 113.050} C_DIS
   LIN {X -1.847, Y 42.265, Z 113.050} C_DIS
   LIN {X -1.604, Y 41.851, Z 113.050} C_DIS
   LIN {X -1.064, Y 40.883, Z 113.050} C_DIS
   LIN {X 0.652, Y 37.848, Z 113.050} C_DIS
   LIN {X 1.278, Y 36.633, Z 113.050} C_DIS
   LIN {X 3.805, Y 31.351, Z 113.050} C_DIS
   LIN {X 4.220, Y 30.520, Z 113.050} C_DIS
   LIN {X 4.452, Y 30.041, Z 113.050} C_DIS
   LIN {X 6.818, Y 24.170, Z 113.050} C_DIS
   LIN {X 6.931, Y 23.892, Z 113.050} C_DIS
   LIN {X 8.505, Y 19.080, Z 113.050} C_DIS
   LIN {X 9.476, Y 16.123, Z 113.050} C_DIS
   LIN {X 9.524, Y 15.926, Z 113.050} C_DIS
   LIN {X 11.986, Y 5.366, Z 113.050} C_DIS
   LIN {X 12.200, Y 3.957, Z 113.050} C_DIS
   LIN {X 13.133, Y -2.551, Z 113.050} C_DIS
   LIN {X 13.365, Y -5.366, Z 113.050} C_DIS
   LIN {X 13.568, Y -7.972, Z 113.050} C_DIS
   LIN {X 13.589, Y -8.520, Z 113.050} C_DIS
   LIN {X 13.700, Y -10.975, Z 113.050} C_DIS
   LIN {X 13.738, Y -13.219, Z 113.050} C_DIS
   LIN {X 13.747, Y -13.937, Z 113.050} C_DIS
   LIN {X 13.732, Y -14.954, Z 113.050} C_DIS
   LIN {X 13.712, Y -17.199, Z 113.050} C_DIS
   LIN {X 13.295, Y -18.924, Z 113.050} C_DIS
   LIN {X 12.921, Y -20.640, Z 113.050} C_DIS
   LIN {X 12.027, Y -22.073, Z 113.050} C_DIS
   LIN {X 11.271, Y -23.141, Z 113.050} C_DIS
   LIN {X 8.813, Y -24.843, Z 113.050} C_DIS
   LIN {X 8.102, Y -25.356, Z 113.050} C_DIS
   LIN {X 7.570, Y -25.489, Z 113.050} C_DIS
   LIN {X 6.360, Y -25.755, Z 113.050} C_DIS
   LIN {X 5.195, Y -26.031, Z 113.050} C_DIS
   LIN {X 3.466, Y -25.964, Z 113.050} C_DIS
   LIN {X 3.283, Y -25.953, Z 113.050} C_DIS
   LIN {X 0.155, Y -24.682, Z 113.050} C_DIS
   LIN {X -0.811, Y -24.221, Z 113.050} C_DIS
   LIN {X -1.605, Y -23.280, Z 113.050} C_DIS
   LIN {X -3.272, Y -21.319, Z 113.050} C_DIS
   LIN {X -4.259, Y -17.909, Z 113.050} C_DIS
   LIN {X -4.303, Y -17.753, Z 113.050} C_DIS
   LIN {X -3.971, Y -14.600, Z 113.050} C_DIS
   LIN {X -3.272, Y -11.899, Z 113.050} C_DIS
   LIN {X -2.988, Y -10.784, Z 113.050} C_DIS
   LIN {X -2.498, Y -8.312, Z 113.050} C_DIS
   LIN {X -2.219, Y -6.940, Z 113.050} C_DIS
   LIN {X -2.157, Y -6.551, Z 113.050} C_DIS
   LIN {X -1.621, Y -2.885, Z 113.050} C_DIS
   LIN {X -1.165, Y 5.286, Z 113.050} C_DIS
   LIN {X -1.157, Y 5.410, Z 113.050} C_DIS
   LIN {X -1.795, Y 15.035, Z 113.050} C_DIS
   LIN {X -1.939, Y 15.904, Z 113.050} C_DIS
   LIN {X -3.420, Y 23.451, Z 113.050} C_DIS
   LIN {X -3.760, Y 24.561, Z 113.050} C_DIS
   LIN {X -5.628, Y 30.585, Z 113.050} C_DIS
   LIN {X -5.753, Y 30.877, Z 113.050} C_DIS
   LIN {X -6.493, Y 32.759, Z 113.050} C_DIS
   LIN {X -6.603, Y 33.033, Z 113.050} C_DIS
   LIN {X -6.662, Y 33.169, Z 113.050} C_DIS
   LIN {X -8.159, Y 36.561, Z 113.050} C_DIS
   LIN {X -8.905, Y 38.085, Z 113.050}
   LaserEnd_Ext()
   LIN {X 12.602, Y -8.820, Z 113.050}
   LaserStart_Ext()
   LIN {X 12.602, Y -17.537, Z 113.050}
   LaserEnd_Ext()
   LIN {X 11.602, Y -20.866, Z 113.050}
   LaserStart_Ext()
   LIN {X 11.602, Y 1.082, Z 113.050}
   LaserEnd_Ext()
   LIN {X 10.602, Y 6.900, Z 113.050}
   LaserStart_Ext()
   LIN {X 10.602, Y -16.464, Z 113.050}
   LaserEnd_Ext()
   LIN {X 10.602, Y -17.517, Z 113.050}
   LaserStart_Ext()
   LIN {X 10.602, Y -22.355, Z 113.050}
   LaserEnd_Ext()
   LIN {X 9.602, Y -23.080, Z 113.050}
   LaserStart_Ext()
   LIN {X 9.602, Y -20.322, Z 113.050}
   LaserEnd_Ext()
   LIN {X 9.602, Y -13.756, Z 113.050}
   LaserStart_Ext()
   LIN {X 9.602, Y 11.189, Z 113.050}
   LaserEnd_Ext()
   LIN {X 8.602, Y 15.478, Z 113.050}
   LaserStart_Ext()
   LIN {X 8.602, Y -12.580, Z 113.050}
   LaserEnd_Ext()
   LIN {X 8.602, Y -21.526, Z 113.050}
   LaserStart_Ext()
   LIN {X 8.602, Y -23.772, Z 113.050}
   LaserEnd_Ext()
   LIN {X 7.602, Y -24.451, Z 113.050}
   LaserStart_Ext()
   LIN {X 7.602, Y -22.150, Z 113.050}
   LaserEnd_Ext()
   LIN {X 7.602, Y -11.842, Z 113.050}
   LaserStart_Ext()
   LIN {X 7.602, Y 18.626, Z 113.050}
   LaserEnd_Ext()
   LIN {X 6.602, Y 21.681, Z 113.050}
   LaserStart_Ext()
   LIN {X 6.602, Y -11.427, Z 113.050}
   LaserEnd_Ext()
   LIN {X 6.602, Y -22.633, Z 113.050}
   LaserStart_Ext()
   LIN {X 6.602, Y -24.678, Z 113.050}
   LaserEnd_Ext()
   LIN {X 5.602, Y -24.907, Z 113.050}
   LaserStart_Ext()
   LIN {X 5.602, Y -22.909, Z 113.050}
   LaserEnd_Ext()
   LIN {X 5.602, Y -11.096, Z 113.050}
   LaserStart_Ext()
   LIN {X 5.602, Y 24.512, Z 113.050}
   LaserEnd_Ext()
   LIN {X 4.602, Y 26.993, Z 113.050}
   LaserStart_Ext()
   LIN {X 4.602, Y -11.137, Z 113.050}
   LaserEnd_Ext()
   LIN {X 4.602, Y -22.939, Z 113.050}
   LaserStart_Ext()
   LIN {X 4.602, Y -25.007, Z 113.050}
   LaserEnd_Ext()
   LIN {X 3.602, Y -24.969, Z 113.050}
   LaserStart_Ext()
   LIN {X 3.602, Y -22.950, Z 113.050}
   LaserEnd_Ext()
   LIN {X 3.602, Y -11.183, Z 113.050}
   LaserStart_Ext()
   LIN {X 3.602, Y 29.474, Z 113.050}
   LaserEnd_Ext()
   LIN {X 2.602, Y 31.549, Z 113.050}
   LaserStart_Ext()
   LIN {X 2.602, Y -11.498, Z 113.050}
   LaserEnd_Ext()
   LIN {X 2.602, Y -22.568, Z 113.050}
   LaserStart_Ext()
   LIN {X 2.602, Y -24.597, Z 113.050}
   LaserEnd_Ext()
   LIN {X 1.602, Y -24.191, Z 113.050}
   LaserStart_Ext()
   LIN {X 1.602, Y -22.155, Z 113.050}
   LaserEnd_Ext()
   LIN {X 1.602, Y -12.014, Z 113.050}
   LaserStart_Ext()
   LIN {X 1.602, Y 33.639, Z 113.050}
   LaserEnd_Ext()
   LIN {X 0.602, Y 35.729, Z 113.050}
   LaserStart_Ext()
   LIN {X 0.602, Y -12.716, Z 113.050}
   LaserEnd_Ext()
   LIN {X 0.602, Y -21.315, Z 113.050}
   LaserStart_Ext()
   LIN {X 0.602, Y -23.784, Z 113.050}
   LaserEnd_Ext()
   LIN {X -0.398, Y -23.159, Z 113.050}
   LaserStart_Ext()
   LIN {X -0.398, Y -20.255, Z 113.050}
   LaserEnd_Ext()
   LIN {X -0.398, Y -13.980, Z 113.050}
   LaserStart_Ext()
   LIN {X -0.398, Y 1.076, Z 113.050}
   LaserEnd_Ext()
   LIN {X -0.398, Y 9.123, Z 113.050}
   LaserStart_Ext()
   LIN {X -0.398, Y 37.673, Z 113.050}
   LaserEnd_Ext()
   LIN {X -1.398, Y 39.443, Z 113.050}
   LaserStart_Ext()
   LIN {X -1.398, Y 18.341, Z 113.050}
   LaserEnd_Ext()
   LIN {X -1.398, Y -7.922, Z 113.050}
   LaserStart_Ext()
   LIN {X -1.398, Y -21.979, Z 113.050}
   LaserEnd_Ext()
   LIN {X -2.398, Y -20.743, Z 113.050}
   LaserStart_Ext()
   LIN {X -2.398, Y -12.515, Z 113.050}
   LaserEnd_Ext()
   LIN {X -2.398, Y 23.437, Z 113.050}
   LaserStart_Ext()
   LIN {X -2.398, Y 41.222, Z 113.050}
   LaserEnd_Ext()
   LIN {X -3.398, Y 42.897, Z 113.050}
   LaserStart_Ext()
   LIN {X -3.398, Y 26.770, Z 113.050}
   LaserEnd_Ext()
   LIN {X -4.398, Y 29.995, Z 113.050}
   LaserStart_Ext()
   LIN {X -4.398, Y 44.493, Z 113.050}
   LaserEnd_Ext()
   LIN {X -5.398, Y 45.685, Z 113.050}
   LaserStart_Ext()
   LIN {X -5.398, Y 32.707, Z 113.050}
   LaserEnd_Ext()
   LIN {X -6.398, Y 35.048, Z 113.050}
   LaserStart_Ext()
   LIN {X -6.398, Y 46.156, Z 113.050}
   LaserEnd_Ext()
   LIN {X -7.398, Y 46.245, Z 113.050}
   LaserStart_Ext()
   LIN {X -7.398, Y 37.281, Z 113.050}
   LaserEnd_Ext()
   LIN {X -8.398, Y 39.308, Z 113.050}
   LaserStart_Ext()
   LIN {X -8.398, Y 45.885, Z 113.050}
   LaserEnd_Ext()
   LIN {X -9.398, Y 45.219, Z 113.050}
   LaserStart_Ext()
   LIN {X -9.398, Y 41.182, Z 113.050}
   LaserEnd_Ext()
   LIN {X -0.187, Y -17.669, Z 113.900}
   LaserStart_Ext()
   LIN {X -0.183, Y -17.512, Z 113.900} C_DIS
   LIN {X 0.199, Y -15.043, Z 113.900} C_DIS
   LIN {X 1.523, Y -13.199, Z 113.900} C_DIS
   LIN {X 1.611, Y -13.121, Z 113.900} C_DIS
   LIN {X 3.507, Y -12.134, Z 113.900} C_DIS
   LIN {X 5.096, Y -12.060, Z 113.900} C_DIS
   LIN {X 5.681, Y -12.031, Z 113.900} C_DIS
   LIN {X 6.343, Y -12.303, Z 113.900} C_DIS
   LIN {X 7.645, Y -12.843, Z 113.900} C_DIS
   LIN {X 8.681, Y -14.061, Z 113.900} C_DIS
   LIN {X 9.296, Y -14.777, Z 113.900} C_DIS
   LIN {X 9.459, Y -15.491, Z 113.900} C_DIS
   LIN {X 9.783, Y -16.932, Z 113.900} C_DIS
   LIN {X 9.336, Y -18.720, Z 113.900} C_DIS
   LIN {X 9.192, Y -19.291, Z 113.900} C_DIS
   LIN {X 8.048, Y -20.671, Z 113.900} C_DIS
   LIN {X 7.868, Y -20.888, Z 113.900} C_DIS
   LIN {X 7.428, Y -21.100, Z 113.900} C_DIS
   LIN {X 5.908, Y -21.838, Z 113.900} C_DIS
   LIN {X 4.932, Y -21.872, Z 113.900} C_DIS
   LIN {X 3.860, Y -21.905, Z 113.900} C_DIS
   LIN {X 2.414, Y -21.313, Z 113.900} C_DIS
   LIN {X 1.945, Y -21.122, Z 113.900} C_DIS
   LIN {X 1.659, Y -20.826, Z 113.900} C_DIS
   LIN {X 0.503, Y -19.620, Z 113.900} C_DIS
   LIN {X -0.053, Y -18.037, Z 113.900} C_DIS
   LIN {X -0.187, Y -17.669, Z 113.900}
   LaserEnd_Ext()
   LIN {X -5.764, Y 30.851, Z 113.900}
   LaserStart_Ext()
   LIN {X -6.467, Y 32.637, Z 113.900} C_DIS
   LIN {X -6.718, Y 33.227, Z 113.900} C_DIS
   LIN {X -7.924, Y 35.935, Z 113.900} C_DIS
   LIN {X -8.255, Y 36.687, Z 113.900} C_DIS
   LIN {X -8.371, Y 36.924, Z 113.900} C_DIS
   LIN {X -9.366, Y 38.916, Z 113.900} C_DIS
   LIN {X -10.119, Y 40.326, Z 113.900} C_DIS
   LIN {X -10.630, Y 41.253, Z 113.900} C_DIS
   LIN {X -10.723, Y 41.420, Z 113.900} C_DIS
   LIN {X -10.809, Y 41.640, Z 113.900} C_DIS
   LIN {X -11.170, Y 42.565, Z 113.900} C_DIS
   LIN {X -11.177, Y 43.617, Z 113.900} C_DIS
   LIN {X -11.181, Y 44.197, Z 113.900} C_DIS
   LIN {X -10.896, Y 44.853, Z 113.900} C_DIS
   LIN {X -10.513, Y 45.720, Z 113.900} C_DIS
   LIN {X -9.666, Y 46.577, Z 113.900} C_DIS
   LIN {X -9.384, Y 46.742, Z 113.900} C_DIS
   LIN {X -8.267, Y 47.253, Z 113.900} C_DIS
   LIN {X -7.606, Y 47.272, Z 113.900} C_DIS
   LIN {X -6.526, Y 47.300, Z 113.900} C_DIS
   LIN {X -5.028, Y 46.646, Z 113.900} C_DIS
   LIN {X -4.935, Y 46.606, Z 113.900} C_DIS
   LIN {X -3.927, Y 45.538, Z 113.900} C_DIS
   LIN {X -3.234, Y 44.454, Z 113.900} C_DIS
   LIN {X -3.128, Y 44.287, Z 113.900} C_DIS
   LIN {X -2.986, Y 44.056, Z 113.900} C_DIS
   LIN {X -2.279, Y 42.895, Z 113.900} C_DIS
   LIN {X -1.756, Y 42.039, Z 113.900} C_DIS
   LIN {X -1.666, Y 41.893, Z 113.900} C_DIS
   LIN {X -1.571, Y 41.724, Z 113.900} C_DIS
   LIN {X 0.728, Y 37.656, Z 113.900} C_DIS
   LIN {X 1.174, Y 36.789, Z 113.900} C_DIS
   LIN {X 2.977, Y 33.022, Z 113.900} C_DIS
   LIN {X 3.946, Y 31.079, Z 113.900} C_DIS
   LIN {X 4.488, Y 29.958, Z 113.900} C_DIS
   LIN {X 6.587, Y 24.750, Z 113.900} C_DIS
   LIN {X 7.034, Y 23.648, Z 113.900} C_DIS
   LIN {X 9.357, Y 16.551, Z 113.900} C_DIS
   LIN {X 9.635, Y 15.643, Z 113.900} C_DIS
   LIN {X 12.089, Y 5.021, Z 113.900} C_DIS
   LIN {X 13.224, Y -2.851, Z 113.900} C_DIS
   LIN {X 13.392, Y -4.901, Z 113.900} C_DIS
   LIN {X 13.568, Y -7.157, Z 113.900} C_DIS
   LIN {X 13.631, Y -7.929, Z 113.900} C_DIS
   LIN {X 13.648, Y -8.141, Z 113.900} C_DIS
   LIN {X 13.670, Y -8.626, Z 113.900} C_DIS
   LIN {X 13.772, Y -10.890, Z 113.900} C_DIS
   LIN {X 13.813, Y -13.362, Z 113.900} C_DIS
   LIN {X 13.825, Y -13.853, Z 113.900} C_DIS
   LIN {X 13.823, Y -14.375, Z 113.900} C_DIS
   LIN {X 13.800, Y -17.115, Z 113.900} C_DIS
   LIN {X 13.052, Y -20.207, Z 113.900} C_DIS
   LIN {X 12.936, Y -20.742, Z 113.900} C_DIS
   LIN {X 12.656, Y -21.190, Z 113.900} C_DIS
   LIN {X 11.212, Y -23.228, Z 113.900} C_DIS
   LIN {X 8.898, Y -24.831, Z 113.900} C_DIS
   LIN {X 8.269, Y -25.259, Z 113.900} C_DIS
   LIN {X 7.194, Y -25.496, Z 113.900} C_DIS
   LIN {X 5.166, Y -25.976, Z 113.900} C_DIS
   LIN {X 3.854, Y -25.925, Z 113.900} C_DIS
   LIN {X 3.220, Y -25.863, Z 113.900} C_DIS
   LIN {X -0.537, Y -24.254, Z 113.900} C_DIS
   LIN {X -0.702, Y -24.180, Z 113.900} C_DIS
   LIN {X -0.851, Y -24.011, Z 113.900} C_DIS
   LIN {X -3.176, Y -21.277, Z 113.900} C_DIS
   LIN {X -3.932, Y -18.666, Z 113.900} C_DIS
   LIN {X -4.214, Y -17.715, Z 113.900} C_DIS
   LIN {X -4.070, Y -16.244, Z 113.900} C_DIS
   LIN {X -3.893, Y -14.560, Z 113.900} C_DIS
   LIN {X -3.534, Y -13.175, Z 113.900} C_DIS
   LIN {X -2.917, Y -10.742, Z 113.900} C_DIS
   LIN {X -2.247, Y -7.366, Z 113.900} C_DIS
   LIN {X -2.178, Y -7.021, Z 113.900} C_DIS
   LIN {X -2.097, Y -6.461, Z 113.900} C_DIS
   LIN {X -1.582, Y -2.941, Z 113.900} C_DIS
   LIN {X -1.215, Y 3.627, Z 113.900} C_DIS
   LIN {X -1.132, Y 4.971, Z 113.900} C_DIS
   LIN {X -1.152, Y 5.971, Z 113.900} C_DIS
   LIN {X -1.728, Y 14.597, Z 113.900} C_DIS
   LIN {X -2.040, Y 16.475, Z 113.900} C_DIS
   LIN {X -3.368, Y 23.244, Z 113.900} C_DIS
   LIN {X -3.940, Y 25.110, Z 113.900} C_DIS
   LIN {X -5.603, Y 30.474, Z 113.900} C_DIS
   LIN {X -5.764, Y 30.851, Z 113.900}
   LaserEnd_Ext()
   LIN {X -9.303, Y 45.522, Z 113.900}
   LaserStart_Ext()
   LIN {X -5.287, Y 45.522, Z 113.900}
   LaserEnd_Ext()
   LIN {X -4.464, Y 44.522, Z 113.900}
   LaserStart_Ext()
   LIN {X -9.949, Y 44.522, Z 113.900}
   LaserEnd_Ext()
   LIN {X -10.176, Y 43.522, Z 113.900}
   LaserStart_Ext()
   LIN {X -3.831, Y 43.522, Z 113.900}
   LaserEnd_Ext()
   LIN {X -3.222, Y 42.522, Z 113.900}
   LaserStart_Ext()
   LIN {X -10.079, Y 42.522, Z 113.900}
   LaserEnd_Ext()
   LIN {X -9.637, Y 41.522, Z 113.900}
   LaserStart_Ext()
   LIN {X -2.612, Y 41.522, Z 113.900}
   LaserEnd_Ext()
   LIN {X -2.041, Y 40.522, Z 113.900}
   LaserStart_Ext()
   LIN {X -9.090, Y 40.522, Z 113.900}
   LaserEnd_Ext()
   LIN {X -8.556, Y 39.522, Z 113.900}
   LaserStart_Ext()
   LIN {X -1.475, Y 39.522, Z 113.900}
   LaserEnd_Ext()
   LIN {X -0.910, Y 38.522, Z 113.900}
   LaserStart_Ext()
   LIN {X -8.052, Y 38.522, Z 113.900}
   LaserEnd_Ext()
   LIN {X -7.552, Y 37.522, Z 113.900}
   LaserStart_Ext()
   LIN {X -0.345, Y 37.522, Z 113.900}
   LaserEnd_Ext()
   LIN {X 0.187, Y 36.522, Z 113.900}
   LaserStart_Ext()
   LIN {X -7.089, Y 36.522, Z 113.900}
   LaserEnd_Ext()
   LIN {X -6.645, Y 35.522, Z 113.900}
   LaserStart_Ext()
   LIN {X 0.672, Y 35.522, Z 113.900}
   LaserEnd_Ext()
   LIN {X 1.151, Y 34.522, Z 113.900}
   LaserStart_Ext()
   LIN {X -6.200, Y 34.522, Z 113.900}
   LaserEnd_Ext()
   LIN {X -5.756, Y 33.522, Z 113.900}
   LaserStart_Ext()
   LIN {X 1.629, Y 33.522, Z 113.900}
   LaserEnd_Ext()
   LIN {X 2.109, Y 32.522, Z 113.900}
   LaserStart_Ext()
   LIN {X -5.347, Y 32.522, Z 113.900}
   LaserEnd_Ext()
   LIN {X -4.954, Y 31.522, Z 113.900}
   LaserStart_Ext()
   LIN {X 2.607, Y 31.522, Z 113.900}
   LaserEnd_Ext()
   LIN {X 3.104, Y 30.522, Z 113.900}
   LaserStart_Ext()
   LIN {X -4.571, Y 30.522, Z 113.900}
   LaserEnd_Ext()
   LIN {X -4.261, Y 29.522, Z 113.900}
   LaserStart_Ext()
   LIN {X 3.586, Y 29.522, Z 113.900}
   LaserEnd_Ext()
   LIN {X 3.989, Y 28.522, Z 113.900}
   LaserStart_Ext()
   LIN {X -3.951, Y 28.522, Z 113.900}
   LaserEnd_Ext()
   LIN {X -3.641, Y 27.522, Z 113.900}
   LaserStart_Ext()
   LIN {X 4.392, Y 27.522, Z 113.900}
   LaserEnd_Ext()
   LIN {X 4.795, Y 26.522, Z 113.900}
   LaserStart_Ext()
   LIN {X -3.331, Y 26.522, Z 113.900}
   LaserEnd_Ext()
   LIN {X -3.021, Y 25.522, Z 113.900}
   LaserStart_Ext()
   LIN {X 5.198, Y 25.522, Z 113.900}
   LaserEnd_Ext()
   LIN {X 5.601, Y 24.522, Z 113.900}
   LaserStart_Ext()
   LIN {X -2.714, Y 24.522, Z 113.900}
   LaserEnd_Ext()
   LIN {X -2.408, Y 23.522, Z 113.900}
   LaserStart_Ext()
   LIN {X 6.006, Y 23.522, Z 113.900}
   LaserEnd_Ext()
   LIN {X 6.350, Y 22.522, Z 113.900}
   LaserStart_Ext()
   LIN {X -2.207, Y 22.522, Z 113.900}
   LaserEnd_Ext()
   LIN {X -2.011, Y 21.522, Z 113.900}
   LaserStart_Ext()
   LIN {X 6.678, Y 21.522, Z 113.900}
   LaserEnd_Ext()
   LIN {X 7.005, Y 20.522, Z 113.900}
   LaserStart_Ext()
   LIN {X -1.815, Y 20.522, Z 113.900}
   LaserEnd_Ext()
   LIN {X -1.618, Y 19.522, Z 113.900}
   LaserStart_Ext()
   LIN {X 7.332, Y 19.522, Z 113.900}
   LaserEnd_Ext()
   LIN {X 7.659, Y 18.522, Z 113.900}
   LaserStart_Ext()
   LIN {X -1.422, Y 18.522, Z 113.900}
   LaserEnd_Ext()
   LIN {X -1.226, Y 17.522, Z 113.900}
   LaserStart_Ext()
   LIN {X 7.987, Y 17.522, Z 113.900}
   LaserEnd_Ext()
   LIN {X 8.314, Y 16.522, Z 113.900}
   LaserStart_Ext()
   LIN {X -1.034, Y 16.522, Z 113.900}
   LaserEnd_Ext()
   LIN {X -0.868, Y 15.522, Z 113.900}
   LaserStart_Ext()
   LIN {X 8.626, Y 15.522, Z 113.900}
   LaserEnd_Ext()
   LIN {X 8.868, Y 14.522, Z 113.900}
   LaserStart_Ext()
   LIN {X -0.721, Y 14.522, Z 113.900}
   LaserEnd_Ext()
   LIN {X -0.654, Y 13.522, Z 113.900}
   LaserStart_Ext()
   LIN {X 9.099, Y 13.522, Z 113.900}
   LaserEnd_Ext()
   LIN {X 9.330, Y 12.522, Z 113.900}
   LaserStart_Ext()
   LIN {X -0.587, Y 12.522, Z 113.900}
   LaserEnd_Ext()
   LIN {X -0.520, Y 11.522, Z 113.900}
   LaserStart_Ext()
   LIN {X 9.561, Y 11.522, Z 113.900}
   LaserEnd_Ext()
   LIN {X 9.792, Y 10.522, Z 113.900}
   LaserStart_Ext()
   LIN {X -0.454, Y 10.522, Z 113.900}
   LaserEnd_Ext()
   LIN {X -0.387, Y 9.522, Z 113.900}
   LaserStart_Ext()
   LIN {X 10.023, Y 9.522, Z 113.900}
   LaserEnd_Ext()
   LIN {X 10.254, Y 8.522, Z 113.900}
   LaserStart_Ext()
   LIN {X -0.320, Y 8.522, Z 113.900}
   LaserEnd_Ext()
   LIN {X -0.254, Y 7.522, Z 113.900}
   LaserStart_Ext()
   LIN {X 10.485, Y 7.522, Z 113.900}
   LaserEnd_Ext()
   LIN {X 10.716, Y 6.522, Z 113.900}
   LaserStart_Ext()
   LIN {X -0.187, Y 6.522, Z 113.900}
   LaserEnd_Ext()
   LIN {X -0.143, Y 5.522, Z 113.900}
   LaserStart_Ext()
   LIN {X 10.947, Y 5.522, Z 113.900}
   LaserEnd_Ext()
   LIN {X 11.156, Y 4.522, Z 113.900}
   LaserStart_Ext()
   LIN {X -0.158, Y 4.522, Z 113.900}
   LaserEnd_Ext()
   LIN {X -0.220, Y 3.522, Z 113.900}
   LaserStart_Ext()
   LIN {X 11.300, Y 3.522, Z 113.900}
   LaserEnd_Ext()
   LIN {X 11.443, Y 2.522, Z 113.900}
   LaserStart_Ext()
   LIN {X -0.275, Y 2.522, Z 113.900}
   LaserEnd_Ext()
   LIN {X -0.331, Y 1.522, Z 113.900}
   LaserStart_Ext()
   LIN {X 11.586, Y 1.522, Z 113.900}
   LaserEnd_Ext()
   LIN {X 11.730, Y 0.522, Z 113.900}
   LaserStart_Ext()
   LIN {X -0.387, Y 0.522, Z 113.900}
   LaserEnd_Ext()
   LIN {X -0.443, Y -0.478, Z 113.900}
   LaserStart_Ext()
   LIN {X 11.873, Y -0.478, Z 113.900}
   LaserEnd_Ext()
   LIN {X 12.017, Y -1.478, Z 113.900}
   LaserStart_Ext()
   LIN {X -0.499, Y -1.478, Z 113.900}
   LaserEnd_Ext()
   LIN {X -0.555, Y -2.478, Z 113.900}
   LaserStart_Ext()
   LIN {X 12.160, Y -2.478, Z 113.900}
   LaserEnd_Ext()
   LIN {X 12.272, Y -3.478, Z 113.900}
   LaserStart_Ext()
   LIN {X -0.650, Y -3.478, Z 113.900}
   LaserEnd_Ext()
   LIN {X -0.796, Y -4.478, Z 113.900}
   LaserStart_Ext()
   LIN {X 12.354, Y -4.478, Z 113.900}
   LaserEnd_Ext()
   LIN {X 12.434, Y -5.478, Z 113.900}
   LaserStart_Ext()
   LIN {X -0.943, Y -5.478, Z 113.900}
   LaserEnd_Ext()
   LIN {X -1.089, Y -6.478, Z 113.900}
   LaserStart_Ext()
   LIN {X 12.512, Y -6.478, Z 113.900}
   LaserEnd_Ext()
   LIN {X 12.591, Y -7.478, Z 113.900}
   LaserStart_Ext()
   LIN {X -1.249, Y -7.478, Z 113.900}
   LaserEnd_Ext()
   LIN {X -1.448, Y -8.478, Z 113.900}
   LaserStart_Ext()
   LIN {X 12.662, Y -8.478, Z 113.900}
   LaserEnd_Ext()
   LIN {X 12.707, Y -9.478, Z 113.900}
   LaserStart_Ext()
   LIN {X -1.646, Y -9.478, Z 113.900}
   LaserEnd_Ext()
   LIN {X -1.845, Y -10.478, Z 113.900}
   LaserStart_Ext()
   LIN {X 12.752, Y -10.478, Z 113.900}
   LaserEnd_Ext()
   LIN {X 12.782, Y -11.478, Z 113.900}
   LaserStart_Ext()
   LIN {X 6.964, Y -11.478, Z 113.900}
   LaserEnd_Ext()
   LIN {X 2.600, Y -11.478, Z 113.900}
   LaserStart_Ext()
   LIN {X -2.072, Y -11.478, Z 113.900}
   LaserEnd_Ext()
   LIN {X -2.326, Y -12.478, Z 113.900}
   LaserStart_Ext()
   LIN {X 0.822, Y -12.478, Z 113.900}
   LaserEnd_Ext()
   LIN {X 8.648, Y -12.478, Z 113.900}
   LaserStart_Ext()
   LIN {X 12.798, Y -12.478, Z 113.900}
   LaserEnd_Ext()
   LIN {X 12.816, Y -13.478, Z 113.900}
   LaserStart_Ext()
   LIN {X 9.499, Y -13.478, Z 113.900}
   LaserEnd_Ext()
   LIN {X 0.091, Y -13.478, Z 113.900}
   LaserStart_Ext()
   LIN {X -2.580, Y -13.478, Z 113.900}
   LaserEnd_Ext()
   LIN {X -2.839, Y -14.478, Z 113.900}
   LaserStart_Ext()
   LIN {X -0.625, Y -14.478, Z 113.900}
   LaserEnd_Ext()
   LIN {X 10.250, Y -14.478, Z 113.900}
   LaserStart_Ext()
   LIN {X 12.823, Y -14.478, Z 113.900}
   LaserEnd_Ext()
   LIN {X 12.814, Y -15.478, Z 113.900}
   LaserStart_Ext()
   LIN {X 10.481, Y -15.478, Z 113.900}
   LaserEnd_Ext()
   LIN {X -0.880, Y -15.478, Z 113.900}
   LaserStart_Ext()
   LIN {X -2.984, Y -15.478, Z 113.900}
   LaserEnd_Ext()
   LIN {X -3.088, Y -16.478, Z 113.900}
   LaserStart_Ext()
   LIN {X -1.035, Y -16.478, Z 113.900}
   LaserEnd_Ext()
   LIN {X 10.706, Y -16.478, Z 113.900}
   LaserStart_Ext()
   LIN {X 12.805, Y -16.478, Z 113.900}
   LaserEnd_Ext()
   LIN {X 12.683, Y -17.478, Z 113.900}
   LaserStart_Ext()
   LIN {X 10.677, Y -17.478, Z 113.900}
   LaserEnd_Ext()
   LIN {X -1.182, Y -17.478, Z 113.900}
   LaserStart_Ext()
   LIN {X -3.186, Y -17.478, Z 113.900}
   LaserEnd_Ext()
   LIN {X -2.945, Y -18.478, Z 113.900}
   LaserStart_Ext()
   LIN {X -0.958, Y -18.478, Z 113.900}
   LaserEnd_Ext()
   LIN {X 10.427, Y -18.478, Z 113.900}
   LaserStart_Ext()
   LIN {X 12.441, Y -18.478, Z 113.900}
   LaserEnd_Ext()
   LIN {X 12.200, Y -19.478, Z 113.900}
   LaserStart_Ext()
   LIN {X 10.176, Y -19.478, Z 113.900}
   LaserEnd_Ext()
   LIN {X -0.607, Y -19.478, Z 113.900}
   LaserStart_Ext()
   LIN {X -2.656, Y -19.478, Z 113.900}
   LaserEnd_Ext()
   LIN {X -2.366, Y -20.478, Z 113.900}
   LaserStart_Ext()
   LIN {X -0.060, Y -20.478, Z 113.900}
   LaserEnd_Ext()
   LIN {X 9.506, Y -20.478, Z 113.900}
   LaserStart_Ext()
   LIN {X 11.922, Y -20.478, Z 113.900}
   LaserEnd_Ext()
   LIN {X 11.226, Y -21.478, Z 113.900}
   LaserStart_Ext()
   LIN {X 8.677, Y -21.478, Z 113.900}
   LaserEnd_Ext()
   LIN {X 0.899, Y -21.478, Z 113.900}
   LaserStart_Ext()
   LIN {X -1.692, Y -21.478, Z 113.900}
   LaserEnd_Ext()
   LIN {X -0.842, Y -22.478, Z 113.900}
   LaserStart_Ext()
   LIN {X 2.621, Y -22.478, Z 113.900}
   LaserEnd_Ext()
   LIN {X 6.879, Y -22.478, Z 113.900}
   LaserStart_Ext()
   LIN {X 10.518, Y -22.478, Z 113.900}
   LaserEnd_Ext()
   LIN {X 9.094, Y -23.478, Z 113.900}
   LaserStart_Ext()
   LIN {X 0.191, Y -23.478, Z 113.900}
   LaserEnd_Ext()
   LIN {X 2.527, Y -24.478, Z 113.900}
   LaserStart_Ext()
   LIN {X 7.163, Y -24.478, Z 113.900}
   LaserEnd_Ext()
   LIN {X 2.041, Y -21.068, Z 114.750}
   LaserStart_Ext()
   LIN {X 0.751, Y -19.733, Z 114.750} C_DIS
   LIN {X 0.593, Y -19.569, Z 114.750} C_DIS
   LIN {X 0.517, Y -19.353, Z 114.750} C_DIS
   LIN {X -0.090, Y -17.678, Z 114.750} C_DIS
   LIN {X -0.074, Y -16.964, Z 114.750} C_DIS
   LIN {X 0.195, Y -15.231, Z 114.750} C_DIS
   LIN {X 1.169, Y -13.874, Z 114.750} C_DIS
   LIN {X 1.537, Y -13.195, Z 114.750} C_DIS
   LIN {X 3.188, Y -12.280, Z 114.750} C_DIS
   LIN {X 3.580, Y -12.075, Z 114.750} C_DIS
   LIN {X 3.891, Y -12.061, Z 114.750} C_DIS
   LIN {X 5.755, Y -11.967, Z 114.750} C_DIS
   LIN {X 7.597, Y -12.725, Z 114.750} C_DIS
   LIN {X 7.720, Y -12.775, Z 114.750} C_DIS
   LIN {X 7.829, Y -12.901, Z 114.750} C_DIS
   LIN {X 9.377, Y -14.704, Z 114.750} C_DIS
   LIN {X 9.846, Y -16.762, Z 114.750} C_DIS
   LIN {X 9.774, Y -17.230, Z 114.750} C_DIS
   LIN {X 9.279, Y -19.227, Z 114.750} C_DIS
   LIN {X 9.060, Y -19.494, Z 114.750} C_DIS
   LIN {X 7.964, Y -20.818, Z 114.750} C_DIS
   LIN {X 7.091, Y -21.246, Z 114.750} C_DIS
   LIN {X 6.005, Y -21.774, Z 114.750} C_DIS
   LIN {X 4.185, Y -21.837, Z 114.750} C_DIS
   LIN {X 3.956, Y -21.846, Z 114.750} C_DIS
   LIN {X 3.805, Y -21.785, Z 114.750} C_DIS
   LIN {X 2.041, Y -21.068, Z 114.750}
   LaserEnd_Ext()
   LIN {X 7.137, Y 23.403, Z 114.750}
   LaserStart_Ext()
   LIN {X 9.183, Y 17.154, Z 114.750} C_DIS
   LIN {X 9.813, Y 15.099, Z 114.750} C_DIS
   LIN {X 12.013, Y 5.572, Z 114.750} C_DIS
   LIN {X 12.232, Y 4.492, Z 114.750} C_DIS
   LIN {X 12.612, Y 1.744, Z 114.750} C_DIS
   LIN {X 13.314, Y -3.152, Z 114.750} C_DIS
   LIN {X 13.420, Y -4.436, Z 114.750} C_DIS
   LIN {X 13.530, Y -5.849, Z 114.750} C_DIS
   LIN {X 13.690, Y -7.815, Z 114.750} C_DIS
   LIN {X 13.704, Y -7.919, Z 114.750} C_DIS
   LIN {X 13.733, Y -8.355, Z 114.750} C_DIS
   LIN {X 13.789, Y -9.591, Z 114.750} C_DIS
   LIN {X 13.844, Y -10.805, Z 114.750} C_DIS
   LIN {X 13.866, Y -12.131, Z 114.750} C_DIS
   LIN {X 13.906, Y -13.767, Z 114.750} C_DIS
   LIN {X 13.900, Y -15.506, Z 114.750} C_DIS
   LIN {X 13.887, Y -17.030, Z 114.750} C_DIS
   LIN {X 13.262, Y -19.616, Z 114.750} C_DIS
   LIN {X 12.983, Y -20.771, Z 114.750} C_DIS
   LIN {X 12.255, Y -21.761, Z 114.750} C_DIS
   LIN {X 11.153, Y -23.316, Z 114.750} C_DIS
   LIN {X 10.046, Y -24.083, Z 114.750} C_DIS
   LIN {X 8.507, Y -25.130, Z 114.750} C_DIS
   LIN {X 8.028, Y -25.236, Z 114.750} C_DIS
   LIN {X 5.137, Y -25.920, Z 114.750} C_DIS
   LIN {X 4.441, Y -25.893, Z 114.750} C_DIS
   LIN {X 3.100, Y -25.762, Z 114.750} C_DIS
   LIN {X 0.719, Y -24.742, Z 114.750} C_DIS
   LIN {X -0.538, Y -24.174, Z 114.750} C_DIS
   LIN {X -1.680, Y -22.882, Z 114.750} C_DIS
   LIN {X -3.080, Y -21.236, Z 114.750} C_DIS
   LIN {X -3.535, Y -19.663, Z 114.750} C_DIS
   LIN {X -4.123, Y -17.676, Z 114.750} C_DIS
   LIN {X -3.823, Y -14.605, Z 114.750} C_DIS
   LIN {X -3.796, Y -14.451, Z 114.750} C_DIS
   LIN {X -2.845, Y -10.700, Z 114.750} C_DIS
   LIN {X -2.373, Y -8.323, Z 114.750} C_DIS
   LIN {X -2.171, Y -7.309, Z 114.750} C_DIS
   LIN {X -1.933, Y -5.658, Z 114.750} C_DIS
   LIN {X -1.543, Y -2.997, Z 114.750} C_DIS
   LIN {X -1.266, Y 1.969, Z 114.750} C_DIS
   LIN {X -1.108, Y 4.533, Z 114.750} C_DIS
   LIN {X -1.146, Y 6.440, Z 114.750} C_DIS
   LIN {X -1.661, Y 14.160, Z 114.750} C_DIS
   LIN {X -2.140, Y 17.046, Z 114.750} C_DIS
   LIN {X -3.316, Y 23.037, Z 114.750} C_DIS
   LIN {X -4.120, Y 25.659, Z 114.750} C_DIS
   LIN {X -5.579, Y 30.364, Z 114.750} C_DIS
   LIN {X -5.776, Y 30.824, Z 114.750} C_DIS
   LIN {X -6.344, Y 32.269, Z 114.750} C_DIS
   LIN {X -6.944, Y 33.678, Z 114.750} C_DIS
   LIN {X -8.196, Y 36.492, Z 114.750} C_DIS
   LIN {X -8.483, Y 37.068, Z 114.750} C_DIS
   LIN {X -8.933, Y 37.957, Z 114.750} C_DIS
   LIN {X -9.424, Y 38.940, Z 114.750} C_DIS
   LIN {X -9.990, Y 39.993, Z 114.750} C_DIS
   LIN {X -10.181, Y 40.348, Z 114.750} C_DIS
   LIN {X -10.360, Y 40.669, Z 114.750} C_DIS
   LIN {X -10.787, Y 41.440, Z 114.750} C_DIS
   LIN {X -11.041, Y 42.087, Z 114.750} C_DIS
   LIN {X -11.240, Y 42.600, Z 114.750} C_DIS
   LIN {X -11.244, Y 43.602, Z 114.750} C_DIS
   LIN {X -11.248, Y 44.234, Z 114.750} C_DIS
   LIN {X -11.052, Y 44.687, Z 114.750} C_DIS
   LIN {X -10.641, Y 45.657, Z 114.750} C_DIS
   LIN {X -10.318, Y 46.015, Z 114.750} C_DIS
   LIN {X -9.683, Y 46.661, Z 114.750} C_DIS
   LIN {X -8.833, Y 47.057, Z 114.750} C_DIS
   LIN {X -8.345, Y 47.280, Z 114.750} C_DIS
   LIN {X -7.120, Y 47.315, Z 114.750} C_DIS
   LIN {X -6.603, Y 47.331, Z 114.750} C_DIS
   LIN {X -6.302, Y 47.201, Z 114.750} C_DIS
   LIN {X -5.010, Y 46.640, Z 114.750} C_DIS
   LIN {X -4.033, Y 45.611, Z 114.750} C_DIS
   LIN {X -3.967, Y 45.525, Z 114.750} C_DIS
   LIN {X -3.197, Y 44.326, Z 114.750} C_DIS
   LIN {X -2.454, Y 43.108, Z 114.750} C_DIS
   LIN {X -1.537, Y 41.618, Z 114.750} C_DIS
   LIN {X -0.571, Y 39.895, Z 114.750} C_DIS
   LIN {X 0.804, Y 37.463, Z 114.750} C_DIS
   LIN {X 1.071, Y 36.945, Z 114.750} C_DIS
   LIN {X 2.148, Y 34.693, Z 114.750} C_DIS
   LIN {X 3.672, Y 31.637, Z 114.750} C_DIS
   LIN {X 4.524, Y 29.876, Z 114.750} C_DIS
   LIN {X 6.357, Y 25.330, Z 114.750} C_DIS
   LIN {X 7.137, Y 23.403, Z 114.750}
   LaserEnd_Ext()
   LIN {X -9.280, Y 40.784, Z 114.750}
   LaserStart_Ext()
   LIN {X -9.280, Y 45.644, Z 114.750}
   LaserEnd_Ext()
   LIN {X -8.280, Y 46.210, Z 114.750}
   LaserStart_Ext()
   LIN {X -8.280, Y 38.887, Z 114.750}
   LaserEnd_Ext()
   LIN {X -7.280, Y 36.893, Z 114.750}
   LaserStart_Ext()
   LIN {X -7.280, Y 46.310, Z 114.750}
   LaserEnd_Ext()
   LIN {X -6.280, Y 46.101, Z 114.750}
   LaserStart_Ext()
   LIN {X -6.280, Y 34.646, Z 114.750}
   LaserEnd_Ext()
   LIN {X -5.280, Y 32.296, Z 114.750}
   LaserStart_Ext()
   LIN {X -5.280, Y 45.472, Z 114.750}
   LaserEnd_Ext()
   LIN {X -4.280, Y 44.162, Z 114.750}
   LaserStart_Ext()
   LIN {X -4.280, Y 29.552, Z 114.750}
   LaserEnd_Ext()
   LIN {X -3.280, Y 26.327, Z 114.750}
   LaserStart_Ext()
   LIN {X -3.280, Y 42.543, Z 114.750}
   LaserEnd_Ext()
   LIN {X -2.280, Y 40.898, Z 114.750}
   LaserStart_Ext()
   LIN {X -2.280, Y 22.950, Z 114.750}
   LaserEnd_Ext()
   LIN {X -2.280, Y -12.539, Z 114.750}
   LaserStart_Ext()
   LIN {X -2.280, Y -20.403, Z 114.750}
   LaserEnd_Ext()
   LIN {X -1.280, Y -21.808, Z 114.750}
   LaserStart_Ext()
   LIN {X -1.280, Y -7.952, Z 114.750}
   LaserEnd_Ext()
   LIN {X -1.280, Y 17.854, Z 114.750}
   LaserStart_Ext()
   LIN {X -1.280, Y 39.117, Z 114.750}
   LaserEnd_Ext()
   LIN {X -0.280, Y 37.348, Z 114.750}
   LaserStart_Ext()
   LIN {X -0.280, Y 8.478, Z 114.750}
   LaserEnd_Ext()
   LIN {X -0.280, Y 1.693, Z 114.750}
   LaserStart_Ext()
   LIN {X -0.280, Y -14.177, Z 114.750}
   LaserEnd_Ext()
   LIN {X -0.280, Y -20.054, Z 114.750}
   LaserStart_Ext()
   LIN {X -0.280, Y -22.956, Z 114.750}
   LaserEnd_Ext()
   LIN {X 0.720, Y -23.645, Z 114.750}
   LaserStart_Ext()
   LIN {X 0.720, Y -21.140, Z 114.750}
   LaserEnd_Ext()
   LIN {X 0.720, Y -12.619, Z 114.750}
   LaserStart_Ext()
   LIN {X 0.720, Y 35.361, Z 114.750}
   LaserEnd_Ext()
   LIN {X 1.720, Y 33.310, Z 114.750}
   LaserStart_Ext()
   LIN {X 1.720, Y -11.950, Z 114.750}
   LaserEnd_Ext()
   LIN {X 1.720, Y -22.017, Z 114.750}
   LaserStart_Ext()
   LIN {X 1.720, Y -24.083, Z 114.750}
   LaserEnd_Ext()
   LIN {X 2.720, Y -24.511, Z 114.750}
   LaserStart_Ext()
   LIN {X 2.720, Y -22.423, Z 114.750}
   LaserEnd_Ext()
   LIN {X 2.720, Y -11.396, Z 114.750}
   LaserStart_Ext()
   LIN {X 2.720, Y 31.305, Z 114.750}
   LaserEnd_Ext()
   LIN {X 3.720, Y 29.196, Z 114.750}
   LaserStart_Ext()
   LIN {X 3.720, Y -11.068, Z 114.750}
   LaserEnd_Ext()
   LIN {X 3.720, Y -22.816, Z 114.750}
   LaserStart_Ext()
   LIN {X 3.720, Y -24.818, Z 114.750}
   LaserEnd_Ext()
   LIN {X 4.720, Y -24.903, Z 114.750}
   LaserStart_Ext()
   LIN {X 4.720, Y -22.819, Z 114.750}
   LaserEnd_Ext()
   LIN {X 4.720, Y -11.018, Z 114.750}
   LaserStart_Ext()
   LIN {X 4.720, Y 26.715, Z 114.750}
   LaserEnd_Ext()
   LIN {X 5.720, Y 24.238, Z 114.750}
   LaserStart_Ext()
   LIN {X 5.720, Y -10.968, Z 114.750}
   LaserEnd_Ext()
   LIN {X 5.720, Y -22.784, Z 114.750}
   LaserStart_Ext()
   LIN {X 5.720, Y -24.754, Z 114.750}
   LaserEnd_Ext()
   LIN {X 6.720, Y -24.518, Z 114.750}
   LaserStart_Ext()
   LIN {X 6.720, Y -22.538, Z 114.750}
   LaserEnd_Ext()
   LIN {X 6.720, Y -11.283, Z 114.750}
   LaserStart_Ext()
   LIN {X 6.720, Y 21.463, Z 114.750}
   LaserEnd_Ext()
   LIN {X 7.720, Y 18.408, Z 114.750}
   LaserStart_Ext()
   LIN {X 7.720, Y -11.694, Z 114.750}
   LaserEnd_Ext()
   LIN {X 7.720, Y -22.051, Z 114.750}
   LaserStart_Ext()
   LIN {X 7.720, Y -24.281, Z 114.750}
   LaserEnd_Ext()
   LIN {X 8.720, Y -23.775, Z 114.750}
   LaserStart_Ext()
   LIN {X 8.720, Y -21.471, Z 114.750}
   LaserEnd_Ext()
   LIN {X 8.720, Y -12.404, Z 114.750}
   LaserStart_Ext()
   LIN {X 8.720, Y 15.251, Z 114.750}
   LaserEnd_Ext()
   LIN {X 9.720, Y 11.057, Z 114.750}
   LaserStart_Ext()
   LIN {X 9.720, Y -13.569, Z 114.750}
   LaserEnd_Ext()
   LIN {X 9.720, Y -20.265, Z 114.750}
   LaserStart_Ext()
   LIN {X 9.720, Y -23.092, Z 114.750}
   LaserEnd_Ext()
   LIN {X 10.720, Y -22.197, Z 114.750}
   LaserStart_Ext()
   LIN {X 10.720, Y -17.571, Z 114.750}
   LaserEnd_Ext()
   LIN {X 10.720, Y -16.099, Z 114.750}
   LaserStart_Ext()
   LIN {X 10.720, Y 6.728, Z 114.750}
   LaserEnd_Ext()
   LIN {X 11.720, Y 0.921, Z 114.750}
   LaserStart_Ext()
   LIN {X 11.720, Y -20.800, Z 114.750}
   LaserEnd_Ext()
   LIN {X 12.720, Y -17.601, Z 114.750}
   LaserStart_Ext()
   LIN {X 12.720, Y -8.200, Z 114.750}
   LaserEnd_Ext()
   LIN {X 8.994, Y -14.090, Z 115.600}
   LaserStart_Ext()
   LIN {X 9.457, Y -14.631, Z 115.600} C_DIS
   LIN {X 9.612, Y -15.311, Z 115.600} C_DIS
   LIN {X 9.951, Y -16.921, Z 115.600} C_DIS
   LIN {X 9.716, Y -17.767, Z 115.600} C_DIS
   LIN {X 9.372, Y -19.152, Z 115.600} C_DIS
   LIN {X 8.588, Y -20.111, Z 115.600} C_DIS
   LIN {X 8.062, Y -20.747, Z 115.600} C_DIS
   LIN {X 6.187, Y -21.667, Z 115.600} C_DIS
   LIN {X 6.047, Y -21.712, Z 115.600} C_DIS
   LIN {X 4.055, Y -21.786, Z 115.600} C_DIS
   LIN {X 2.658, Y -21.225, Z 115.600} C_DIS
   LIN {X 2.137, Y -21.013, Z 115.600} C_DIS
   LIN {X 1.655, Y -20.514, Z 115.600} C_DIS
   LIN {X 0.687, Y -19.518, Z 115.600} C_DIS
   LIN {X 0.397, Y -18.763, Z 115.600} C_DIS
   LIN {X 0.008, Y -17.688, Z 115.600} C_DIS
   LIN {X 0.035, Y -16.417, Z 115.600} C_DIS
   LIN {X 0.190, Y -15.418, Z 115.600} C_DIS
   LIN {X 0.751, Y -14.637, Z 115.600} C_DIS
   LIN {X 1.502, Y -13.250, Z 115.600} C_DIS
   LIN {X 2.975, Y -12.434, Z 115.600} C_DIS
   LIN {X 3.656, Y -12.017, Z 115.600} C_DIS
   LIN {X 4.959, Y -11.947, Z 115.600} C_DIS
   LIN {X 5.829, Y -11.903, Z 115.600} C_DIS
   LIN {X 6.447, Y -12.157, Z 115.600} C_DIS
   LIN {X 7.798, Y -12.705, Z 115.600} C_DIS
   LIN {X 8.994, Y -14.090, Z 115.600}
   LaserEnd_Ext()
   LIN {X 0.967, Y 37.101, Z 115.600}
   LaserStart_Ext()
   LIN {X 1.320, Y 36.364, Z 115.600} C_DIS
   LIN {X 3.398, Y 32.196, Z 115.600} C_DIS
   LIN {X 4.561, Y 29.793, Z 115.600} C_DIS
   LIN {X 6.126, Y 25.909, Z 115.600} C_DIS
   LIN {X 7.241, Y 23.159, Z 115.600} C_DIS
   LIN {X 9.009, Y 17.756, Z 115.600} C_DIS
   LIN {X 9.990, Y 14.556, Z 115.600} C_DIS
   LIN {X 11.921, Y 6.199, Z 115.600} C_DIS
   LIN {X 12.358, Y 4.034, Z 115.600} C_DIS
   LIN {X 13.122, Y -1.477, Z 115.600} C_DIS
   LIN {X 13.405, Y -3.453, Z 115.600} C_DIS
   LIN {X 13.448, Y -3.971, Z 115.600} C_DIS
   LIN {X 13.492, Y -4.541, Z 115.600} C_DIS
   LIN {X 13.749, Y -7.701, Z 115.600} C_DIS
   LIN {X 13.771, Y -7.869, Z 115.600} C_DIS
   LIN {X 13.818, Y -8.570, Z 115.600} C_DIS
   LIN {X 13.908, Y -10.556, Z 115.600} C_DIS
   LIN {X 13.915, Y -10.720, Z 115.600} C_DIS
   LIN {X 13.918, Y -10.900, Z 115.600} C_DIS
   LIN {X 13.988, Y -13.681, Z 115.600} C_DIS
   LIN {X 13.977, Y -16.638, Z 115.600} C_DIS
   LIN {X 13.974, Y -16.946, Z 115.600} C_DIS
   LIN {X 13.848, Y -17.468, Z 115.600} C_DIS
   LIN {X 13.057, Y -20.740, Z 115.600} C_DIS
   LIN {X 11.177, Y -23.295, Z 115.600} C_DIS
   LIN {X 11.085, Y -23.408, Z 115.600} C_DIS
   LIN {X 8.803, Y -24.963, Z 115.600} C_DIS
   LIN {X 8.604, Y -25.051, Z 115.600} C_DIS
   LIN {X 6.520, Y -25.530, Z 115.600} C_DIS
   LIN {X 5.108, Y -25.865, Z 115.600} C_DIS
   LIN {X 2.980, Y -25.660, Z 115.600} C_DIS
   LIN {X 1.974, Y -25.230, Z 115.600} C_DIS
   LIN {X -0.375, Y -24.169, Z 115.600} C_DIS
   LIN {X -2.508, Y -21.753, Z 115.600} C_DIS
   LIN {X -2.984, Y -21.194, Z 115.600} C_DIS
   LIN {X -3.138, Y -20.660, Z 115.600} C_DIS
   LIN {X -4.033, Y -17.637, Z 115.600} C_DIS
   LIN {X -3.813, Y -15.381, Z 115.600} C_DIS
   LIN {X -3.731, Y -14.481, Z 115.600} C_DIS
   LIN {X -3.347, Y -12.921, Z 115.600} C_DIS
   LIN {X -2.773, Y -10.658, Z 115.600} C_DIS
   LIN {X -2.500, Y -9.281, Z 115.600} C_DIS
   LIN {X -2.165, Y -7.596, Z 115.600} C_DIS
   LIN {X -1.768, Y -4.856, Z 115.600} C_DIS
   LIN {X -1.505, Y -3.053, Z 115.600} C_DIS
   LIN {X -1.317, Y 0.311, Z 115.600} C_DIS
   LIN {X -1.083, Y 4.095, Z 115.600} C_DIS
   LIN {X -1.140, Y 6.909, Z 115.600} C_DIS
   LIN {X -1.594, Y 13.723, Z 115.600} C_DIS
   LIN {X -2.241, Y 17.617, Z 115.600} C_DIS
   LIN {X -3.264, Y 22.831, Z 115.600} C_DIS
   LIN {X -4.299, Y 26.207, Z 115.600} C_DIS
   LIN {X -5.554, Y 30.254, Z 115.600} C_DIS
   LIN {X -5.787, Y 30.798, Z 115.600} C_DIS
   LIN {X -6.221, Y 31.901, Z 115.600} C_DIS
   LIN {X -7.169, Y 34.129, Z 115.600} C_DIS
   LIN {X -8.102, Y 36.225, Z 115.600} C_DIS
   LIN {X -8.740, Y 37.507, Z 115.600} C_DIS
   LIN {X -9.458, Y 38.926, Z 115.600} C_DIS
   LIN {X -9.813, Y 39.577, Z 115.600} C_DIS
   LIN {X -10.240, Y 40.370, Z 115.600} C_DIS
   LIN {X -10.536, Y 40.901, Z 115.600} C_DIS
   LIN {X -10.849, Y 41.461, Z 115.600} C_DIS
   LIN {X -11.313, Y 42.657, Z 115.600} C_DIS
   LIN {X -11.315, Y 43.074, Z 115.600} C_DIS
   LIN {X -11.346, Y 43.878, Z 115.600} C_DIS
   LIN {X -11.146, Y 44.706, Z 115.600} C_DIS
   LIN {X -10.779, Y 45.574, Z 115.600} C_DIS
   LIN {X -9.904, Y 46.540, Z 115.600} C_DIS
   LIN {X -9.770, Y 46.676, Z 115.600} C_DIS
   LIN {X -9.286, Y 46.902, Z 115.600} C_DIS
   LIN {X -8.455, Y 47.299, Z 115.600} C_DIS
   LIN {X -7.764, Y 47.330, Z 115.600} C_DIS
   LIN {X -6.677, Y 47.363, Z 115.600} C_DIS
   LIN {X -5.170, Y 46.712, Z 115.600} C_DIS
   LIN {X -5.042, Y 46.632, Z 115.600} C_DIS
   LIN {X -4.068, Y 45.614, Z 115.600} C_DIS
   LIN {X -3.266, Y 44.365, Z 115.600} C_DIS
   LIN {X -3.152, Y 44.178, Z 115.600} C_DIS
   LIN {X -1.408, Y 41.344, Z 115.600} C_DIS
   LIN {X 0.430, Y 38.067, Z 115.600} C_DIS
   LIN {X 0.880, Y 37.271, Z 115.600} C_DIS
   LIN {X 0.967, Y 37.101, Z 115.600}
   LaserEnd_Ext()
   LIN {X 7.147, Y -24.360, Z 115.600}
   LaserStart_Ext()
   LIN {X 2.484, Y -24.360, Z 115.600}
   LaserEnd_Ext()
   LIN {X 0.265, Y -23.360, Z 115.600}
   LaserStart_Ext()
   LIN {X 9.380, Y -23.360, Z 115.600}
   LaserEnd_Ext()
   LIN {X 10.624, Y -22.360, Z 115.600}
   LaserStart_Ext()
   LIN {X 7.044, Y -22.360, Z 115.600}
   LaserEnd_Ext()
   LIN {X 2.802, Y -22.360, Z 115.600}
   LaserStart_Ext()
   LIN {X -0.638, Y -22.360, Z 115.600}
   LaserEnd_Ext()
   LIN {X -1.521, Y -21.360, Z 115.600}
   LaserStart_Ext()
   LIN {X 1.081, Y -21.360, Z 115.600}
   LaserEnd_Ext()
   LIN {X 8.852, Y -21.360, Z 115.600}
   LaserStart_Ext()
   LIN {X 11.359, Y -21.360, Z 115.600}
   LaserEnd_Ext()
   LIN {X 12.095, Y -20.360, Z 115.600}
   LaserStart_Ext()
   LIN {X 9.676, Y -20.360, Z 115.600}
   LaserEnd_Ext()
   LIN {X 0.111, Y -20.360, Z 115.600}
   LaserStart_Ext()
   LIN {X -2.184, Y -20.360, Z 115.600}
   LaserEnd_Ext()
   LIN {X -2.480, Y -19.360, Z 115.600}
   LaserStart_Ext()
   LIN {X -0.445, Y -19.360, Z 115.600}
   LaserEnd_Ext()
   LIN {X 10.351, Y -19.360, Z 115.600}
   LaserStart_Ext()
   LIN {X 12.361, Y -19.360, Z 115.600}
   LaserEnd_Ext()
   LIN {X 12.603, Y -18.360, Z 115.600}
   LaserStart_Ext()
   LIN {X 10.599, Y -18.360, Z 115.600}
   LaserEnd_Ext()
   LIN {X -0.812, Y -18.360, Z 115.600}
   LaserStart_Ext()
   LIN {X -2.776, Y -18.360, Z 115.600}
   LaserEnd_Ext()
   LIN {X -3.002, Y -17.360, Z 115.600}
   LaserStart_Ext()
   LIN {X -0.985, Y -17.360, Z 115.600}
   LaserEnd_Ext()
   LIN {X 10.867, Y -17.360, Z 115.600}
   LaserStart_Ext()
   LIN {X 12.845, Y -17.360, Z 115.600}
   LaserEnd_Ext()
   LIN {X 12.978, Y -16.360, Z 115.600}
   LaserStart_Ext()
   LIN {X 10.855, Y -16.360, Z 115.600}
   LaserEnd_Ext()
   LIN {X -0.961, Y -16.360, Z 115.600}
   LaserStart_Ext()
   LIN {X -2.904, Y -16.360, Z 115.600}
   LaserEnd_Ext()
   LIN {X -2.807, Y -15.360, Z 115.600}
   LaserStart_Ext()
   LIN {X -0.813, Y -15.360, Z 115.600}
   LaserEnd_Ext()
   LIN {X 10.645, Y -15.360, Z 115.600}
   LaserStart_Ext()
   LIN {X 12.981, Y -15.360, Z 115.600}
   LaserEnd_Ext()
   LIN {X 12.985, Y -14.360, Z 115.600}
   LaserStart_Ext()
   LIN {X 10.419, Y -14.360, Z 115.600}
   LaserEnd_Ext()
   LIN {X -0.281, Y -14.360, Z 115.600}
   LaserStart_Ext()
   LIN {X -2.672, Y -14.360, Z 115.600}
   LaserEnd_Ext()
   LIN {X -2.426, Y -13.360, Z 115.600}
   LaserStart_Ext()
   LIN {X 0.305, Y -13.360, Z 115.600}
   LaserEnd_Ext()
   LIN {X 9.684, Y -13.360, Z 115.600}
   LaserStart_Ext()
   LIN {X 12.979, Y -13.360, Z 115.600}
   LaserEnd_Ext()
   LIN {X 12.954, Y -12.360, Z 115.600}
   LaserStart_Ext()
   LIN {X 8.821, Y -12.360, Z 115.600}
   LaserEnd_Ext()
   LIN {X 1.045, Y -12.360, Z 115.600}
   LaserStart_Ext()
   LIN {X -2.173, Y -12.360, Z 115.600}
   LaserEnd_Ext()
   LIN {X -1.920, Y -11.360, Z 115.600}
   LaserStart_Ext()
   LIN {X 2.813, Y -11.360, Z 115.600}
   LaserEnd_Ext()
   LIN {X 7.143, Y -11.360, Z 115.600}
   LaserStart_Ext()
   LIN {X 12.929, Y -11.360, Z 115.600}
   LaserEnd_Ext()
   LIN {X 12.898, Y -10.360, Z 115.600}
   LaserStart_Ext()
   LIN {X -1.695, Y -10.360, Z 115.600}
   LaserEnd_Ext()
   LIN {X -1.496, Y -9.360, Z 115.600}
   LaserStart_Ext()
   LIN {X 12.852, Y -9.360, Z 115.600}
   LaserEnd_Ext()
   LIN {X 12.801, Y -8.360, Z 115.600}
   LaserStart_Ext()
   LIN {X -1.297, Y -8.360, Z 115.600}
   LaserEnd_Ext()
   LIN {X -1.120, Y -7.360, Z 115.600}
   LaserStart_Ext()
   LIN {X 12.718, Y -7.360, Z 115.600}
   LaserEnd_Ext()
   LIN {X 12.637, Y -6.360, Z 115.600}
   LaserStart_Ext()
   LIN {X -0.975, Y -6.360, Z 115.600}
   LaserEnd_Ext()
   LIN {X -0.831, Y -5.360, Z 115.600}
   LaserStart_Ext()
   LIN {X 12.555, Y -5.360, Z 115.600}
   LaserEnd_Ext()
   LIN {X 12.475, Y -4.360, Z 115.600}
   LaserStart_Ext()
   LIN {X -0.685, Y -4.360, Z 115.600}
   LaserEnd_Ext()
   LIN {X -0.539, Y -3.360, Z 115.600}
   LaserStart_Ext()
   LIN {X 12.381, Y -3.360, Z 115.600}
   LaserEnd_Ext()
   LIN {X 12.238, Y -2.360, Z 115.600}
   LaserStart_Ext()
   LIN {X -0.464, Y -2.360, Z 115.600}
   LaserEnd_Ext()
   LIN {X -0.408, Y -1.360, Z 115.600}
   LaserStart_Ext()
   LIN {X 12.096, Y -1.360, Z 115.600}
   LaserEnd_Ext()
   LIN {X 11.957, Y -0.360, Z 115.600}
   LaserStart_Ext()
   LIN {X -0.353, Y -0.360, Z 115.600}
   LaserEnd_Ext()
   LIN {X -0.295, Y 0.640, Z 115.600}
   LaserStart_Ext()
   LIN {X 11.819, Y 0.640, Z 115.600}
   LaserEnd_Ext()
   LIN {X 11.680, Y 1.640, Z 115.600}
   LaserStart_Ext()
   LIN {X -0.233, Y 1.640, Z 115.600}
   LaserEnd_Ext()
   LIN {X -0.171, Y 2.640, Z 115.600}
   LaserStart_Ext()
   LIN {X 11.542, Y 2.640, Z 115.600}
   LaserEnd_Ext()
   LIN {X 11.403, Y 3.640, Z 115.600}
   LaserStart_Ext()
   LIN {X -0.109, Y 3.640, Z 115.600}
   LaserEnd_Ext()
   LIN {X -0.094, Y 4.640, Z 115.600}
   LaserStart_Ext()
   LIN {X 11.215, Y 4.640, Z 115.600}
   LaserEnd_Ext()
   LIN {X 11.013, Y 5.640, Z 115.600}
   LaserStart_Ext()
   LIN {X -0.114, Y 5.640, Z 115.600}
   LaserEnd_Ext()
   LIN {X -0.134, Y 6.640, Z 115.600}
   LaserStart_Ext()
   LIN {X 10.792, Y 6.640, Z 115.600}
   LaserEnd_Ext()
   LIN {X 10.561, Y 7.640, Z 115.600}
   LaserStart_Ext()
   LIN {X -0.186, Y 7.640, Z 115.600}
   LaserEnd_Ext()
   LIN {X -0.253, Y 8.640, Z 115.600}
   LaserStart_Ext()
   LIN {X 10.331, Y 8.640, Z 115.600}
   LaserEnd_Ext()
   LIN {X 10.100, Y 9.640, Z 115.600}
   LaserStart_Ext()
   LIN {X -0.320, Y 9.640, Z 115.600}
   LaserEnd_Ext()
   LIN {X -0.386, Y 10.640, Z 115.600}
   LaserStart_Ext()
   LIN {X 9.869, Y 10.640, Z 115.600}
   LaserEnd_Ext()
   LIN {X 9.638, Y 11.640, Z 115.600}
   LaserStart_Ext()
   LIN {X -0.453, Y 11.640, Z 115.600}
   LaserEnd_Ext()
   LIN {X -0.520, Y 12.640, Z 115.600}
   LaserStart_Ext()
   LIN {X 9.407, Y 12.640, Z 115.600}
   LaserEnd_Ext()
   LIN {X 9.176, Y 13.640, Z 115.600}
   LaserStart_Ext()
   LIN {X -0.587, Y 13.640, Z 115.600}
   LaserEnd_Ext()
   LIN {X -0.733, Y 14.640, Z 115.600}
   LaserStart_Ext()
   LIN {X 8.919, Y 14.640, Z 115.600}
   LaserEnd_Ext()
   LIN {X 8.612, Y 15.640, Z 115.600}
   LaserStart_Ext()
   LIN {X -0.899, Y 15.640, Z 115.600}
   LaserEnd_Ext()
   LIN {X -1.065, Y 16.640, Z 115.600}
   LaserStart_Ext()
   LIN {X 8.305, Y 16.640, Z 115.600}
   LaserEnd_Ext()
   LIN {X 7.995, Y 17.640, Z 115.600}
   LaserStart_Ext()
   LIN {X -1.231, Y 17.640, Z 115.600}
   LaserEnd_Ext()
   LIN {X -1.423, Y 18.640, Z 115.600}
   LaserStart_Ext()
   LIN {X 7.668, Y 18.640, Z 115.600}
   LaserEnd_Ext()
   LIN {X 7.340, Y 19.640, Z 115.600}
   LaserStart_Ext()
   LIN {X -1.619, Y 19.640, Z 115.600}
   LaserEnd_Ext()
   LIN {X -1.815, Y 20.640, Z 115.600}
   LaserStart_Ext()
   LIN {X 7.013, Y 20.640, Z 115.600}
   LaserEnd_Ext()
   LIN {X 6.686, Y 21.640, Z 115.600}
   LaserStart_Ext()
   LIN {X -2.011, Y 21.640, Z 115.600}
   LaserEnd_Ext()
   LIN {X -2.208, Y 22.640, Z 115.600}
   LaserStart_Ext()
   LIN {X 6.358, Y 22.640, Z 115.600}
   LaserEnd_Ext()
   LIN {X 5.967, Y 23.640, Z 115.600}
   LaserStart_Ext()
   LIN {X -2.466, Y 23.640, Z 115.600}
   LaserEnd_Ext()
   LIN {X -2.773, Y 24.640, Z 115.600}
   LaserStart_Ext()
   LIN {X 5.561, Y 24.640, Z 115.600}
   LaserEnd_Ext()
   LIN {X 5.156, Y 25.640, Z 115.600}
   LaserStart_Ext()
   LIN {X -3.079, Y 25.640, Z 115.600}
   LaserEnd_Ext()
   LIN {X -3.387, Y 26.640, Z 115.600}
   LaserStart_Ext()
   LIN {X 4.753, Y 26.640, Z 115.600}
   LaserEnd_Ext()
   LIN {X 4.350, Y 27.640, Z 115.600}
   LaserStart_Ext()
   LIN {X -3.697, Y 27.640, Z 115.600}
   LaserEnd_Ext()
   LIN {X -4.007, Y 28.640, Z 115.600}
   LaserStart_Ext()
   LIN {X 3.947, Y 28.640, Z 115.600}
   LaserEnd_Ext()
   LIN {X 3.524, Y 29.640, Z 115.600}
   LaserStart_Ext()
   LIN {X -4.317, Y 29.640, Z 115.600}
   LaserEnd_Ext()
   LIN {X -4.632, Y 30.640, Z 115.600}
   LaserStart_Ext()
   LIN {X 3.040, Y 30.640, Z 115.600}
   LaserEnd_Ext()
   LIN {X 2.556, Y 31.640, Z 115.600}
   LaserStart_Ext()
   LIN {X -5.043, Y 31.640, Z 115.600}
   LaserEnd_Ext()
   LIN {X -5.448, Y 32.640, Z 115.600}
   LaserStart_Ext()
   LIN {X 2.059, Y 32.640, Z 115.600}
   LaserEnd_Ext()
   LIN {X 1.560, Y 33.640, Z 115.600}
   LaserStart_Ext()
   LIN {X -5.874, Y 33.640, Z 115.600}
   LaserEnd_Ext()
   LIN {X -6.302, Y 34.640, Z 115.600}
   LaserStart_Ext()
   LIN {X 1.062, Y 34.640, Z 115.600}
   LaserEnd_Ext()
   LIN {X 0.563, Y 35.640, Z 115.600}
   LaserStart_Ext()
   LIN {X -6.747, Y 35.640, Z 115.600}
   LaserEnd_Ext()
   LIN {X -7.192, Y 36.640, Z 115.600}
   LaserStart_Ext()
   LIN {X 0.079, Y 36.640, Z 115.600}
   LaserEnd_Ext()
   LIN {X -0.477, Y 37.640, Z 115.600}
   LaserStart_Ext()
   LIN {X -7.689, Y 37.640, Z 115.600}
   LaserEnd_Ext()
   LIN {X -8.193, Y 38.640, Z 115.600}
   LaserStart_Ext()
   LIN {X -1.038, Y 38.640, Z 115.600}
   LaserEnd_Ext()
   LIN {X -1.599, Y 39.640, Z 115.600}
   LaserStart_Ext()
   LIN {X -8.709, Y 39.640, Z 115.600}
   LaserEnd_Ext()
   LIN {X -9.250, Y 40.640, Z 115.600}
   LaserStart_Ext()
   LIN {X -2.160, Y 40.640, Z 115.600}
   LaserEnd_Ext()
   LIN {X -2.765, Y 41.640, Z 115.600}
   LaserStart_Ext()
   LIN {X -9.804, Y 41.640, Z 115.600}
   LaserEnd_Ext()
   LIN {X -10.234, Y 42.640, Z 115.600}
   LaserStart_Ext()
   LIN {X -3.380, Y 42.640, Z 115.600}
   LaserEnd_Ext()
   LIN {X -3.995, Y 43.640, Z 115.600}
   LaserStart_Ext()
   LIN {X -10.336, Y 43.640, Z 115.600}
   LaserEnd_Ext()
   LIN {X -10.088, Y 44.640, Z 115.600}
   LaserStart_Ext()
   LIN {X -4.631, Y 44.640, Z 115.600}
   LaserEnd_Ext()
   LIN {X -5.477, Y 45.640, Z 115.600}
   LaserStart_Ext()
   LIN {X -9.370, Y 45.640, Z 115.600}
   LaserEnd_Ext()
   LIN {X 9.767, Y -15.717, Z 116.450}
   LaserStart_Ext()
   LIN {X 10.036, Y -16.993, Z 116.450} C_DIS
   LIN {X 9.547, Y -18.752, Z 116.450} C_DIS
   LIN {X 9.466, Y -19.077, Z 116.450} C_DIS
   LIN {X 8.415, Y -20.363, Z 116.450} C_DIS
   LIN {X 8.160, Y -20.676, Z 116.450} C_DIS
   LIN {X 6.203, Y -21.644, Z 116.450} C_DIS
   LIN {X 4.888, Y -21.699, Z 116.450} C_DIS
   LIN {X 4.155, Y -21.726, Z 116.450} C_DIS
   LIN {X 3.192, Y -21.340, Z 116.450} C_DIS
   LIN {X 2.235, Y -20.958, Z 116.450} C_DIS
   LIN {X 1.649, Y -20.360, Z 116.450} C_DIS
   LIN {X 0.781, Y -19.467, Z 116.450} C_DIS
